	out 5 "открыть ЗДЭ02.13" <= #1228.outputOpen
	out 6 "закрыть ЗДЭ02.13" <= #1228.outputClose
	out 7 "авария открытия ЗДЭ02.13" <= #1228.errorToOpen
	#1229 OR(panTestValvesFS020201, #1230.regenFilterOUT)
	out 8 "авария закрытия ЗДЭ02.13" <= #1228.errorToClose
	#1230 FS020201manager:FilterQueueManager(input: pin 1, filterAlarm: #1231, regenFilterStatus: pin 3, alarmReset: pin 4, startNextLoop: pin 5)
	#1231 OR(alarmZD021319, pin 2, pin 11, pin 12)
	#1232 OR(#1228.errorToOpen, #1228.errorToClose, #1234.errorToOpen, #1234.errorToClose)
	#1233 alarmZD021319 <= #1232
	out 3 "ФС02.02.01 промыт" <= #1230.regenerated
	out 4 "не удалось промыть" <= #1230.failToRegen
	#1234 ZD0219:SimpleValve(inputOpen: #1229, inputClose: NOT #1229, statusOpen: pin 8, statusClose: pin 9, reset: pin 4, timeToOpenClose: pin 10)
	out 9 "открыть ЗДЭ02.19" <= #1234.outputOpen
	out 10 "закрыть ЗДЭ02.19" <= #1234.outputClose
	out 11 "авария открытия ЗДЭ02.19" <= #1234.errorToOpen
	out 12 "авария закрытия ЗДЭ02.19" <= #1234.errorToClose
END_MACRO
#1235 DD2_DO.10 <= #1227.out 2
#1236 regeneratedFS020201 <= #1227.out 3
#1237 filterFailToRegen020201 <= #1227.out 4
#1238 DD3_DO.8 <= #1227.out 5
#1239 DD3_DO.9 <= #1227.out 6
#1240 errorToOpenZD0213 <= #1227.out 7
#1241 errorToCloseZD0213 <= #1227.out 8
#1242 DD3_DO.20 <= #1227.out 9
#1243 DD3_DO.21 <= #1227.out 10
#1244 errorToOpenZD0219 <= #1227.out 11
#1245 errorToCloseZD0219 <= #1227.out 12
#1246 MACRO управление промывкой фильтра ФС02.02.02(pin 1 "сигнал на промывку": #1227.out 1, pin 2 "авария фильтра": DD7_DI.3, pin 3 "подтверждение промывки": DD7_DI.2, pin 4 "сброс аварий": alarmReset, pin 5 "начать очередь снова": filterStartNewQueue, pin 6 "ЗДЭ02.14 открыта": DD8_DI.10, pin 7 "ЗДЭ02.14 закрыта": DD8_DI.11, pin 8 "ЗДЭ02.20 открыта": DD8_DI.22, pin 9 "ЗДЭ02.20 закрыта": DD8_DI.23, pin 10 "время движения ЗДЭ": timeToOpenCloseValve, pin 11 "авария питания ЗДЭ02.14": DD9_DI.17, pin 12 "авария питания ЗДЭ02.20": DD9_DI.23)
	(* <- выход использовать в / последнем фильтре для / начала очереди заново *)
	(* если открыт = промывка *)
	(* если открыт = фильтрация *)
	out 1 "следующий в очереди" <= #1249.output
	out 2 "промыть ФС02.02.02" <= #1248
	#1247 ZD0214:SimpleValve(inputOpen: NOT #1248, inputClose: #1248, statusOpen: pin 6, statusClose: pin 7, reset: pin 4, timeToOpenClose: pin 10)
	out 5 "открыть ЗДЭ02.14" <= #1247.outputOpen
	out 6 "закрыть ЗДЭ02.14" <= #1247.outputClose
	out 7 "авария открытия ЗДЭ02.14" <= #1247.errorToOpen
	#1248 OR(panTestValvesFS020202, #1249.regenFilterOUT)
	out 8 "авария закрытия ЗДЭ02.14" <= #1247.errorToClose
	#1249 FS020202manager:FilterQueueManager(input: pin 1, filterAlarm: #1250, regenFilterStatus: pin 3, alarmReset: pin 4, startNextLoop: pin 5)
	#1250 OR(alarmZD021420, pin 2, pin 11, pin 12)
	#1251 OR(#1247.errorToOpen, #1247.errorToClose, #1253.errorToOpen, #1253.errorToClose)
	#1252 alarmZD021420 <= #1251
	out 3 "ФС02.02.02 промыт" <= #1249.regenerated
	out 4 "не удалось промыть" <= #1249.failToRegen
	#1253 ZD0220:SimpleValve(inputOpen: #1248, inputClose: NOT #1248, statusOpen: pin 8, statusClose: pin 9, reset: pin 4, timeToOpenClose: pin 10)
	out 9 "открыть ЗДЭ02.20" <= #1253.outputOpen
	out 10 "закрыть ЗДЭ02.20" <= #1253.outputClose
	out 11 "авария открытия ЗДЭ02.20" <= #1253.errorToOpen
	out 12 "авария закрытия ЗДЭ02.20" <= #1253.errorToClose
END_MACRO
#1254 DD2_DO.11 <= #1246.out 2
#1255 regeneratedFS020202 <= #1246.out 3
#1256 filterFailToRegen020202 <= #1246.out 4
#1257 DD3_DO.10 <= #1246.out 5
#1258 DD3_DO.11 <= #1246.out 6
#1259 errorToOpenZD0214 <= #1246.out 7
#1260 errorToCloseZD0214 <= #1246.out 8
#1261 DD3_DO.22 <= #1246.out 9
#1262 DD3_DO.23 <= #1246.out 10
#1263 errorToOpenZD0220 <= #1246.out 11
#1264 errorToCloseZD0220 <= #1246.out 12
#1265 MACRO управление промывкой фильтра ФС02.02.03(pin 1 "сигнал на промывку": #1246.out 1, pin 2 "авария фильтра": DD7_DI.5, pin 3 "подтверждение промывки": DD7_DI.4, pin 4 "сброс аварий": alarmReset, pin 5 "начать очередь снова": filterStartNewQueue, pin 6 "ЗДЭ02.15 открыта": DD8_DI.12, pin 7 "ЗДЭ02.15 закрыта": DD8_DI.13, pin 8 "ЗДЭ02.21 открыта": DD8_DI.24, pin 9 "ЗДЭ02.21 закрыта": DD8_DI.25, pin 10 "время движения ЗДЭ": timeToOpenCloseValve, pin 11 "авария питания ЗДЭ02.15": DD9_DI.18, pin 12 "ааврия питания ЗДЭ02.21": DD9_DI.24)
	(* <- выход использовать в / последнем фильтре для / начала очереди заново *)
	(* если открыт = промывка *)
	(* если открыт = фильтрация *)
	out 1 "следующий в очереди" <= #1268.output
	out 2 "промыть ФС02.02.03" <= #1267
	#1266 ZD0215:SimpleValve(inputOpen: NOT #1267, inputClose: #1267, statusOpen: pin 6, statusClose: pin 7, reset: pin 4, timeToOpenClose: pin 10)
	out 5 "открыть ЗДЭ02.15" <= #1266.outputOpen
	out 6 "закрыть ЗДЭ02.15" <= #1266.outputClose
	out 7 "авария открытия ЗДЭ02.15" <= #1266.errorToOpen
	#1267 OR(panTestValvesFS020203, #1268.regenFilterOUT)
	out 8 "авария закрытия ЗДЭ02.15" <= #1266.errorToClose
	#1268 FS020203manager:FilterQueueManager(input: pin 1, filterAlarm: #1269, regenFilterStatus: pin 3, alarmReset: pin 4, startNextLoop: pin 5)
	#1269 OR(alarmZD021521, pin 2, pin 11, pin 12)
	#1270 OR(#1266.errorToOpen, #1266.errorToClose, #1272.errorToOpen, #1272.errorToClose)
	#1271 alarmZD021521 <= #1270
	out 3 "ФС02.02.03 промыт" <= #1268.regenerated
	out 4 "не удалось промыть" <= #1268.failToRegen
	#1272 ZD0221:SimpleValve(inputOpen: #1267, inputClose: NOT #1267, statusOpen: pin 8, statusClose: pin 9, reset: pin 4, timeToOpenClose: pin 10)
	out 9 "открыть ЗДЭ02.21" <= #1272.outputOpen
	out 10 "закрыть ЗДЭ02.21" <= #1272.outputClose
	out 11 "авария открытия ЗДЭ02.21" <= #1272.errorToOpen
	out 12 "авария закрытия ЗДЭ02.21" <= #1272.errorToClose
END_MACRO
#1273 DD2_DO.12 <= #1265.out 2
#1274 regeneratedFS020203 <= #1265.out 3
#1275 filterFailToRegen020203 <= #1265.out 4
#1276 DD3_DO.12 <= #1265.out 5
#1277 DD3_DO.13 <= #1265.out 6
#1278 errorToOpenZD0215 <= #1265.out 7
#1279 errorToCloseZD0215 <= #1265.out 8
#1280 DD3_DO.24 <= #1265.out 9
#1281 DD3_DO.25 <= #1265.out 10
#1282 errorToOpenZD0221 <= #1265.out 11
#1283 errorToCloseZD0221 <= #1265.out 12
#1284 MACRO управление промывкой фильтра ФС02.02.04(pin 1 "сигнал на промывку": #1265.out 1, pin 2 "авария фильтра": DD7_DI.7, pin 3 "подтверждение промывки": DD7_DI.6, pin 4 "сброс аварий": alarmReset, pin 5 "начать очередь снова": filterStartNewQueue, pin 6 "ЗДЭ02.16 открыта": DD8_DI.14, pin 7 "ЗДЭ02.16 закрыта": DD8_DI.15, pin 8 "ЗДЭ02.22 открыта": DD8_DI.26, pin 9 "ЗДЭ02.22 закрыта": DD8_DI.27, pin 10 "время движения ЗДЭ": timeToOpenCloseValve, pin 11 "авария питания ЗДЭ02.16": DD9_DI.19, pin 12 "авария питания ЗДЭ02.22": DD9_DI.25)
	(* <- выход использовать в / последнем фильтре для / начала очереди заново *)
	(* если открыт = промывка *)
	(* если открыт = фильтрация *)
	out 1 "следующий в очереди" <= #1287.output
	out 2 "промыть ФС02.02.04" <= #1286
	#1285 ZD0216:SimpleValve(inputOpen: NOT #1286, inputClose: #1286, statusOpen: pin 6, statusClose: pin 7, reset: pin 4, timeToOpenClose: pin 10)
	out 5 "открыть ЗДЭ02.16" <= #1285.outputOpen
	out 6 "закрыть ЗДЭ02.16" <= #1285.outputClose
	out 7 "авария открытия ЗДЭ02.16" <= #1285.errorToOpen
	#1286 OR(panTestValvesFS020204, #1287.regenFilterOUT)
	out 8 "авария закрытия ЗДЭ02.16" <= #1285.errorToClose
	#1287 FS020204manager:FilterQueueManager(input: pin 1, filterAlarm: #1288, regenFilterStatus: pin 3, alarmReset: pin 4, startNextLoop: pin 5)
	#1288 OR(alarmZD021622, pin 2, pin 11, pin 12)
	#1289 OR(#1285.errorToOpen, #1285.errorToClose, #1291.errorToOpen, #1291.errorToClose)
	#1290 alarmZD021622 <= #1289
	out 3 "ФС02.02.04 промыт" <= #1287.regenerated
	out 4 "не удалось промыть" <= #1287.failToRegen
	#1291 ZD0222:SimpleValve(inputOpen: #1286, inputClose: NOT #1286, statusOpen: pin 8, statusClose: pin 9, reset: pin 4, timeToOpenClose: pin 10)
	out 9 "открыть ЗДЭ02.22" <= #1291.outputOpen
	out 10 "закрыть ЗДЭ02.22" <= #1291.outputClose
	out 11 "авария открытия ЗДЭ02.22" <= #1291.errorToOpen
	out 12 "авария закрытия ЗДЭ02.22" <= #1291.errorToClose
END_MACRO
#1292 DD2_DO.13 <= #1284.out 2
#1293 regeneratedFS020204 <= #1284.out 3
#1294 filterFailToRegen020204 <= #1284.out 4
#1295 DD3_DO.14 <= #1284.out 5
#1296 DD3_DO.15 <= #1284.out 6
#1297 errorToOpenZD0216 <= #1284.out 7
#1298 errorToCloseZD0216 <= #1284.out 8
#1299 DD3_DO.26 <= #1284.out 9
#1300 DD3_DO.27 <= #1284.out 10
#1301 errorToOpenZD0222 <= #1284.out 11
#1302 errorToCloseZD0222 <= #1284.out 12
#1303 MACRO управление промывкой фильтра ФС02.02.05(pin 1 "сигнал на промывку": #1284.out 1, pin 2 "авария фильтра": DD7_DI.9, pin 3 "подтверждение промывки": DD7_DI.8, pin 4 "сброс аварий": alarmReset, pin 5 "начать очередь снова": filterStartNewQueue, pin 6 "ЗДЭ02.17 открыта": DD8_DI.16, pin 7 "ЗДЭ02.17 закрыта": DD8_DI.17, pin 8 "ЗДЭ02.23 открыта": DD8_DI.28, pin 9 "ЗДЭ02.23 закрыта": DD8_DI.29, pin 10 "время движения ЗДЭ": timeToOpenCloseValve, pin 11 "авария питания ЗДЭ02.17": DD9_DI.20, pin 12 "авария питания ЗДЭ02.23": DD9_DI.26)
	(* <- выход использовать в / последнем фильтре для / начала очереди заново *)
	(* если открыт = промывка *)
	(* если открыт = фильтрация *)
	out 1 "следующий в очереди" <= #1306.output
	out 2 "промыть ФС02.02.05" <= #1305
	#1304 ZD0217:SimpleValve(inputOpen: NOT #1305, inputClose: #1305, statusOpen: pin 6, statusClose: pin 7, reset: pin 4, timeToOpenClose: pin 10)
	out 5 "открыть ЗДЭ02.17" <= #1304.outputOpen
	out 6 "закрыть ЗДЭ02.17" <= #1304.outputClose
	out 7 "авария открытия ЗДЭ02.17" <= #1304.errorToOpen
	#1305 OR(panTestValvesFS020205, #1306.regenFilterOUT)
	out 8 "авария закрытия ЗДЭ02.17" <= #1304.errorToClose
	#1306 FS020205manager:FilterQueueManager(input: pin 1, filterAlarm: #1307, regenFilterStatus: pin 3, alarmReset: pin 4, startNextLoop: pin 5)
	#1307 OR(alarmZD021723, pin 2, pin 11, pin 12)
	#1308 OR(#1304.errorToOpen, #1304.errorToClose, #1310.errorToOpen, #1310.errorToClose)
	#1309 alarmZD021723 <= #1308
	out 3 "ФС02.02.05 промыт" <= #1306.regenerated
	out 4 "не удалось промыть" <= #1306.failToRegen
	#1310 ZD0223:SimpleValve(inputOpen: #1305, inputClose: NOT #1305, statusOpen: pin 8, statusClose: pin 9, reset: pin 4, timeToOpenClose: pin 10)
	out 9 "открыть ЗДЭ02.23" <= #1310.outputOpen
	out 10 "закрыть ЗДЭ02.23" <= #1310.outputClose
	out 11 "авария открытия ЗДЭ02.23" <= #1310.errorToOpen
	out 12 "авария закрытия ЗДЭ02.23" <= #1310.errorToClose
END_MACRO
#1311 DD2_DO.14 <= #1303.out 2
#1312 regeneratedFS020205 <= #1303.out 3
#1313 filterFailToRegen020205 <= #1303.out 4
#1314 DD3_DO.16 <= #1303.out 5
#1315 DD3_DO.17 <= #1303.out 6
#1316 errorToOpenZD0217 <= #1303.out 7
#1317 errorToCloseZD0217 <= #1303.out 8
#1318 DD3_DO.28 <= #1303.out 9
#1319 DD3_DO.29 <= #1303.out 10
#1320 errorToOpenZD0223 <= #1303.out 11
#1321 errorToCloseZD0223 <= #1303.out 12
#1322 MACRO управление промывкой фильтра ФС02.02.06(pin 1 "сигнал на промывку": #1303.out 1, pin 2 "авария фильтра": DD7_DI.11, pin 3 "подтверждение промывки": DD7_DI.10, pin 4 "сброс аварий": alarmReset, pin 5 "начать очередь снова": filterStartNewQueue, pin 6 "ЗДЭ02.18 открыта": DD8_DI.18, pin 7 "ЗДЭ02.18 закрыта": DD8_DI.19, pin 8 "ЗДЭ02.24 открыта": DD8_DI.30, pin 9 "ЗДЭ02.24 закрыта": DD8_DI.31, pin 10 "время движения ЗДЭ": timeToOpenCloseValve, pin 11 "авария питания ЗДЭ02.18": DD9_DI.21, pin 12 "авария питания ЗДЭ02.24": DD9_DI.27)
	(* если открыт = промывка *)
	(* если открыт = фильтрация *)
	out 1 "промыть ФС02.02.06" <= #1324
	#1323 ZD0218:SimpleValve(inputOpen: NOT #1324, inputClose: #1324, statusOpen: pin 6, statusClose: pin 7, reset: pin 4, timeToOpenClose: pin 10)
	out 4 "открыть ЗДЭ02.18" <= #1323.outputOpen
	out 5 "закрыть ЗДЭ02.18" <= #1323.outputClose
	out 6 "авария открытия ЗДЭ02.18" <= #1323.errorToOpen
	#1324 OR(panTestValvesFS020206, #1325.regenFilterOUT)
	out 7 "авария закрытия ЗДЭ02.18" <= #1323.errorToClose
	#1325 FS020206manager:FilterQueueManager(input: pin 1, filterAlarm: #1326, regenFilterStatus: pin 3, alarmReset: pin 4, startNextLoop: pin 5)
	#1326 OR(alarmZD021824, pin 2, pin 11, pin 12)
	#1327 OR(#1323.errorToOpen, #1323.errorToClose, #1329.errorToOpen, #1329.errorToClose)
	#1328 alarmZD021824 <= #1327
	out 2 "ФС02.02.06 промыт" <= #1325.regenerated
	out 3 "не удалось промыть" <= #1325.failToRegen
	out 12 "начать очередь снова" <= #1325.regenFinished
	#1329 ZD0224:SimpleValve(inputOpen: #1324, inputClose: NOT #1324, statusOpen: pin 8, statusClose: pin 9, reset: pin 4, timeToOpenClose: pin 10)
	out 8 "открыть ЗДЭ02.24" <= #1329.outputOpen
	out 9 "закрыть ЗДЭ02.24" <= #1329.outputClose
	out 10 "авария открытия ЗДЭ02.24" <= #1329.errorToOpen
	out 11 "авария закрытия ЗДЭ02.24" <= #1329.errorToClose
END_MACRO
#1330 DD2_DO.15 <= #1322.out 1
#1331 regeneratedFS020206 <= #1322.out 2
#1332 filterFailToRegen020206 <= #1322.out 3
#1333 DD3_DO.18 <= #1322.out 4
#1334 DD3_DO.19 <= #1322.out 5
#1335 errorToOpenZD0218 <= #1322.out 6
#1336 errorToCloseZD0218 <= #1322.out 7
#1337 DD3_DO.30 <= #1322.out 8
#1338 DD3_DO.31 <= #1322.out 9
#1339 errorToOpenZD0224 <= #1322.out 10
#1340 errorToCloseZD0224 <= #1322.out 11
#1341 filterStartNewQueue <= #1322.out 12
_END_CFC_
END_PROGRAM

(* POU DosingPumpProportional, CFC *)
FUNCTION_BLOCK DosingPumpProportional
VAR_INPUT
	flowValue: REAL;		(*текущее значение мгновенного расхода, кубометров в час.*)
	setMinPumpDosingValue: REAL := 0;		(*задание минимальной производительности доз.насоса.
По умолчанию, если ничего не подключено ко входу, равно нулю.*)
	setMaxPumpDosingValue: REAL;		(*задание максимальной производительности доз.насоса, в мл/мин*)
	minOutputValue: REAL := 4;		(*минимальное значение выходного сигнала.
По умолчанию, если ничего не подключено ко входу, равно 4.*)
	maxOutputValue: REAL := 20;		(*Максимально значение выходного сигнала.
			По умолчанию, если ничего не подключено ко входу, равно 20.*)
	setKoeffProportionality: REAL;		(*Задание мл на кубометр (коэф.пропорциональности между расходом и дозированием)*)
	minFlowToStart: REAL := 10;		(*Минимальное значение расхода для подачи сигнала на начало дозирования.
			По умолчанию, если ничего не подключено ко входу, равно 10 кубометров в час.*)
END_VAR
VAR_OUTPUT
	outputValue: REAL;		(*Выходной сигнал на дозирующий насос.*)
	dosingError: BOOL;		(*Ошибка производительности дозирования (неверно заданы значения производительности насоса, производительность доз.насоса не соответствует расходу.*)
	startDosingPump: BOOL;		(*Сигнал на запуск дозирующего насоса.*)
END_VAR
VAR
	linearTransformator: LIN_TRAFO;		(*получает на вход значение из указанного диапазона, ставит на выходе пропорциональное значение из другого диапазона.*)
END_VAR
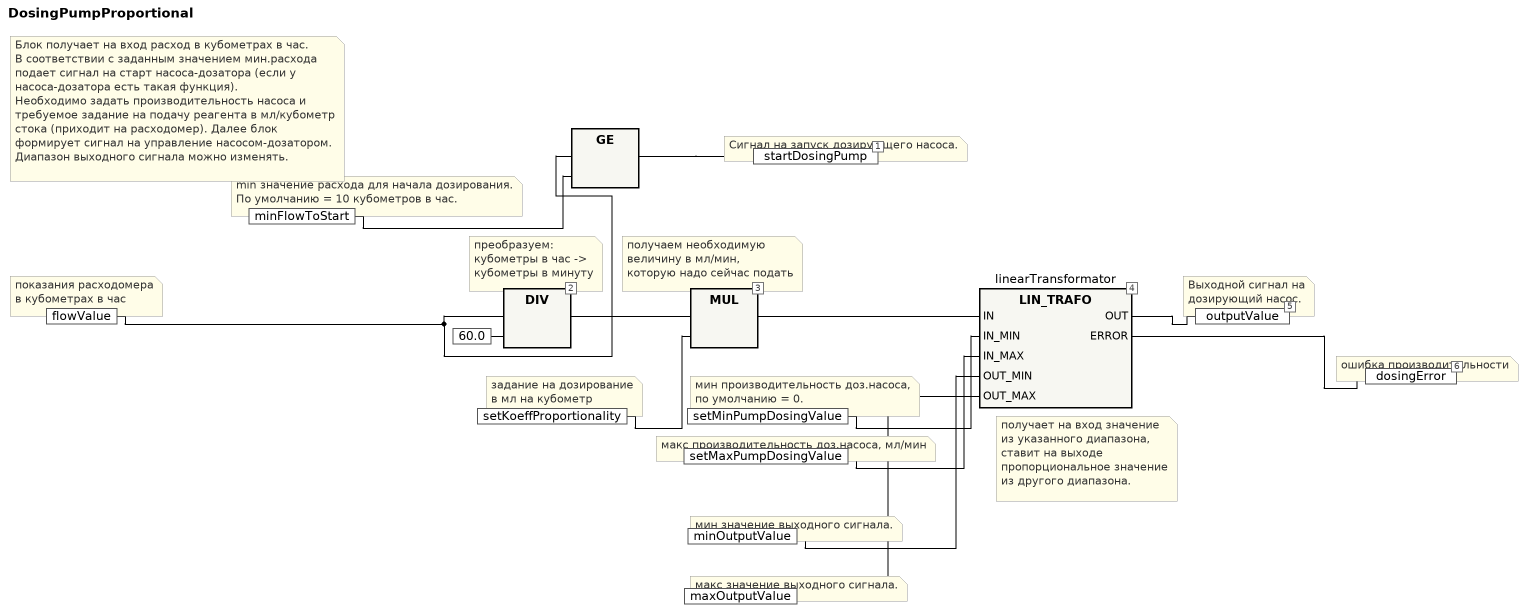
_CFC_ (* Continuous Function Chart, elements in execution order *)
(* Сигнал на запуск дозирующего насоса. *)
(* min значение расхода для начала дозирования. / По умолчанию = 10 кубометров в час. *)
(* макс производительность доз.насоса, мл/мин *)
(* мин производительность доз.насоса, / по умолчанию = 0. *)
(* получаем необходимую / величину в мл/мин, / которую надо сейчас подать *)
(* задание на дозирование / в мл на кубометр *)
(* показания расходомера / в кубометрах в час *)
(* преобразуем: / кубометры в час -> / кубометры в минуту *)
(* мин значение выходного сигнала. *)
(* макс значение выходного сигнала. *)
(* Выходной сигнал на / дозирующий насос. *)
(* ошибка производительности *)
(* получает на вход значение / из указанного диапазона, / ставит на выходе / пропорциональное значение / из другого диапазона. *)
(* Блок получает на вход расход в кубометрах в час. / В соответствии с заданным значением мин.расхода подает сигнал на старт насоса-дозатора (если у насоса-дозатора есть такая функция). / Необходимо задать производительность насоса и требуемое задание на подачу реагента в мл/кубометр стока (приходит на расходомер). Далее блок формирует сигнал на управление насосом-дозатором. / Диапазон выходного сигнала можно изменять. *)
#0 GE(flowValue, minFlowToStart)
#1 startDosingPump <= #0
#2 DIV(flowValue, 60.0)
#3 MUL(#2, setKoeffProportionality)
#4 linearTransformator:LIN_TRAFO(IN: #3, IN_MIN: setMinPumpDosingValue, IN_MAX: setMaxPumpDosingValue, OUT_MIN: minOutputValue, OUT_MAX: maxOutputValue)
#5 outputValue <= #4.OUT
#6 dosingError <= #4.ERROR
_END_CFC_
(* the same logic as Structured Text *)
(* Сигнал на запуск дозирующего насоса. *)
(* min значение расхода для начала дозирования. / По умолчанию = 10 кубометров в час. *)
(* макс производительность доз.насоса, мл/мин *)
(* мин производительность доз.насоса, / по умолчанию = 0. *)
(* получаем необходимую / величину в мл/мин, / которую надо сейчас подать *)
(* задание на дозирование / в мл на кубометр *)
(* показания расходомера / в кубометрах в час *)
(* преобразуем: / кубометры в час -> / кубометры в минуту *)
(* мин значение выходного сигнала. *)
(* макс значение выходного сигнала. *)
(* Выходной сигнал на / дозирующий насос. *)
(* ошибка производительности *)
(* получает на вход значение / из указанного диапазона, / ставит на выходе / пропорциональное значение / из другого диапазона. *)
(* Блок получает на вход расход в кубометрах в час. / В соответствии с заданным значением мин.расхода подает сигнал на старт насоса-дозатора (если у насоса-дозатора есть такая функция). / Необходимо задать производительность насоса и требуемое задание на подачу реагента в мл/кубометр стока (приходит на расходомер). Далее блок формирует сигнал на управление насосом-дозатором. / Диапазон выходного сигнала можно изменять. *)
startDosingPump := flowValue >= minFlowToStart;
linearTransformator(IN := (flowValue / 60.0) * setKoeffProportionality, IN_MIN := setMinPumpDosingValue, IN_MAX := setMaxPumpDosingValue, OUT_MIN := minOutputValue, OUT_MAX := maxOutputValue);
outputValue := linearTransformator.OUT;
dosingError := linearTransformator.ERROR;
END_FUNCTION_BLOCK

(* POU choosePumpRegime, CFC *)
FUNCTION_BLOCK choosePumpRegime
VAR
	pump1RStrig: RS;		(*Триггер-защелка выбора режима с главным первым насосом.*)
	pump2RStrig: RS;		(*Триггер-защелка выбора режима с главным вторым насосом.*)
	byCounterRStrig: RS;		(*Триггер-защелка выбора режима с запуском по количеству включений.*)
	byWorkTimeRStrig: RS;		(*Триггер-защелка выбора режима с запуском по наработке.*)
	Pump1MainDetector: R_TRIG;		(*Детектор переднего фронта включения режима, когда главный насос - первый.
			Для сброса остальных значений.*)
	Pump2MainDetector: R_TRIG;		(*Детектор переднего фронта включения режима, когда главный насос - второй.
			Для сброса остальных значений.*)
	ByCounterDetector: R_TRIG;		(*Детектор переднего фронта включения режима по количеству включений.
			Для сброса остальных значений.*)
	ByWorkTimeDetector: R_TRIG;		(*Детектор переднего фронта включения режима по наработке.
			Для сброса остальных значений.*)
END_VAR
VAR_INPUT
	start: BOOL;		(*Сигнал на включение насоса.
			Активируется выход согласно выбранного режима.*)
	pump1Main: BOOL;		(*Режим: первый насос главный, второй - резервный.*)
	pump2Main: BOOL;		(*Режим: второй насос главный, первый - резервный.*)
	byCounter: BOOL;		(*Режим: запуск по количеству включений.
			Включится с меньшим количеством стартов.*)
	byWorkTime: BOOL;		(*Режим: запуск по наработке.
			Включится насос с меньшей наработкой.*)
END_VAR
VAR_OUTPUT
	pump1MainActive: BOOL;		(*Активный режим: первый насос главный.*)
	pump2MainActive: BOOL;		(*Активный режим: второй насос главный.*)
	byCounterActive: BOOL;		(*Активный режим: включение по количеству запусков.*)
	byWorkTimeActive: BOOL;		(*Активный режим: по наработке.*)
	startPump1: BOOL;		(*Запуск первого насоса как главного (основного).*)
	startPump2: BOOL;		(*Запуск второго насоса как главного (основного).*)
	startByCounter: BOOL;		(*Запуск насоса по количеству стартов.
			Запустится с меньшим. Если одинаково, то - первый.*)
	startByWorkTime: BOOL;		(*Запуск по наработке.
			Включится с меньшей. Если одинаково, то - первый.*)
END_VAR
VAR (* helpers for the ST form of the networks *)
	_en62 : BOOL;
	_t62 : BOOL;
	_en72 : BOOL;
	_t72 : BOOL;
	_en78 : BOOL;
	_t78 : BOOL;
	_en84 : BOOL;
	_t84 : BOOL;
END_VAR
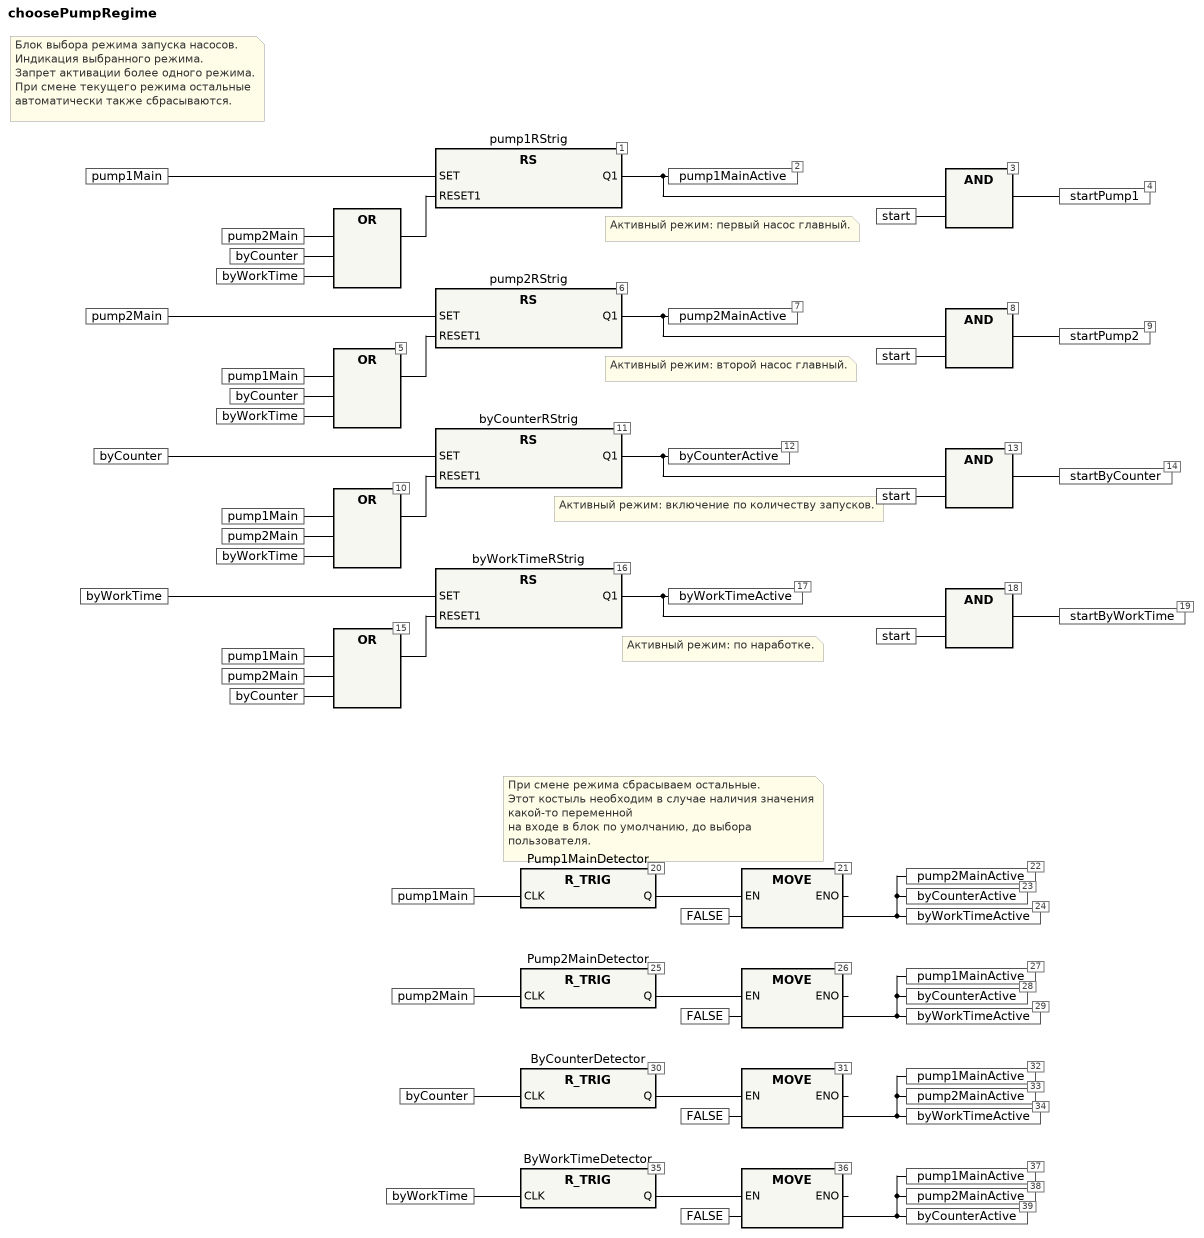
_CFC_ (* Continuous Function Chart, elements in execution order *)
(* Блок выбора режима запуска насосов. / Индикация выбранного режима. / Запрет активации более одного режима. / При смене текущего режима остальные автоматически также сбрасываются. *)
(* Активный режим: первый насос главный. *)
(* Активный режим: включение по количеству запусков. *)
(* Активный режим: по наработке. *)
(* Активный режим: второй насос главный. *)
(* При смене режима сбрасываем остальные. / Этот костыль необходим в случае наличия значения какой-то переменной / на входе в блок по умолчанию, до выбора пользователя. *)
#0 OR(pump2Main, byCounter, byWorkTime)
#1 pump1RStrig:RS(SET: pump1Main, RESET1: #0)
#2 pump1MainActive <= #1.Q1
#3 AND(#1.Q1, start)
#4 startPump1 <= #3
#5 OR(pump1Main, byCounter, byWorkTime)
#6 pump2RStrig:RS(SET: pump2Main, RESET1: #5)
#7 pump2MainActive <= #6.Q1
#8 AND(#6.Q1, start)
#9 startPump2 <= #8
#10 OR(pump1Main, pump2Main, byWorkTime)
#11 byCounterRStrig:RS(SET: byCounter, RESET1: #10)
#12 byCounterActive <= #11.Q1
#13 AND(#11.Q1, start)
#14 startByCounter <= #13
#15 OR(pump1Main, pump2Main, byCounter)
#16 byWorkTimeRStrig:RS(SET: byWorkTime, RESET1: #15)
#17 byWorkTimeActive <= #16.Q1
#18 AND(#16.Q1, start)
#19 startByWorkTime <= #18
#20 Pump1MainDetector:R_TRIG(CLK: pump1Main)
#21 MOVE(EN: #20.Q, FALSE)
#22 pump2MainActive <= #21
#23 byCounterActive <= #21
#24 byWorkTimeActive <= #21
#25 Pump2MainDetector:R_TRIG(CLK: pump2Main)
#26 MOVE(EN: #25.Q, FALSE)
#27 pump1MainActive <= #26
#28 byCounterActive <= #26
#29 byWorkTimeActive <= #26
#30 ByCounterDetector:R_TRIG(CLK: byCounter)
#31 MOVE(EN: #30.Q, FALSE)
#32 pump1MainActive <= #31
#33 pump2MainActive <= #31
#34 byWorkTimeActive <= #31
#35 ByWorkTimeDetector:R_TRIG(CLK: byWorkTime)
#36 MOVE(EN: #35.Q, FALSE)
#37 pump1MainActive <= #36
#38 pump2MainActive <= #36
#39 byCounterActive <= #36
_END_CFC_
(* the same logic as Structured Text *)
(* Блок выбора режима запуска насосов. / Индикация выбранного режима. / Запрет активации более одного режима. / При смене текущего режима остальные автоматически также сбрасываются. *)
(* Активный режим: первый насос главный. *)
(* Активный режим: включение по количеству запусков. *)
(* Активный режим: по наработке. *)
(* Активный режим: второй насос главный. *)
(* При смене режима сбрасываем остальные. / Этот костыль необходим в случае наличия значения какой-то переменной / на входе в блок по умолчанию, до выбора пользователя. *)
pump1RStrig(SET := pump1Main, RESET1 := pump2Main OR byCounter OR byWorkTime);
pump1MainActive := pump1RStrig.Q1;
startPump1 := pump1RStrig.Q1 AND start;
pump2RStrig(SET := pump2Main, RESET1 := pump1Main OR byCounter OR byWorkTime);
pump2MainActive := pump2RStrig.Q1;
startPump2 := pump2RStrig.Q1 AND start;
byCounterRStrig(SET := byCounter, RESET1 := pump1Main OR pump2Main OR byWorkTime);
byCounterActive := byCounterRStrig.Q1;
startByCounter := byCounterRStrig.Q1 AND start;
byWorkTimeRStrig(SET := byWorkTime, RESET1 := pump1Main OR pump2Main OR byCounter);
byWorkTimeActive := byWorkTimeRStrig.Q1;
startByWorkTime := byWorkTimeRStrig.Q1 AND start;
Pump1MainDetector(CLK := pump1Main);
_en62 := Pump1MainDetector.Q;
IF _en62 THEN _t62 := FALSE; END_IF;
IF _en62 THEN pump2MainActive := _t62; END_IF;
IF _en62 THEN byCounterActive := _t62; END_IF;
IF _en62 THEN byWorkTimeActive := _t62; END_IF;
Pump2MainDetector(CLK := pump2Main);
_en72 := Pump2MainDetector.Q;
IF _en72 THEN _t72 := FALSE; END_IF;
IF _en72 THEN pump1MainActive := _t72; END_IF;
IF _en72 THEN byCounterActive := _t72; END_IF;
IF _en72 THEN byWorkTimeActive := _t72; END_IF;
ByCounterDetector(CLK := byCounter);
_en78 := ByCounterDetector.Q;
IF _en78 THEN _t78 := FALSE; END_IF;
IF _en78 THEN pump1MainActive := _t78; END_IF;
IF _en78 THEN pump2MainActive := _t78; END_IF;
IF _en78 THEN byWorkTimeActive := _t78; END_IF;
ByWorkTimeDetector(CLK := byWorkTime);
_en84 := ByWorkTimeDetector.Q;
IF _en84 THEN _t84 := FALSE; END_IF;
IF _en84 THEN pump1MainActive := _t84; END_IF;
IF _en84 THEN pump2MainActive := _t84; END_IF;
IF _en84 THEN byCounterActive := _t84; END_IF;
END_FUNCTION_BLOCK

(* POU TwoPumpManager, CFC *)
FUNCTION_BLOCK TwoPumpManager
VAR_INPUT
	startStopPump1: BOOL;		(*Сигнал на пуск/стоп первого насоса.*)
	startStopPump2: BOOL;		(*Сигнал на пуск/стоп второго насоса.*)
	alarmPump1: BOOL;		(*Сигнал "авария" на первом насосе.*)
	alarmPump2: BOOL;		(*Сигнал "авария" на втором насосе.*)
	alarmReset: BOOL;		(*Сброс аварии.*)

	counterStart: BOOL;		(*Запуск насоса с меньшим количеством включений.*)
	Pump1ResetCounter: BOOL;		(*Сброс счетчика количества включений первого насоса.
Сбрасывается также автоматически при достижении счетчиком значения ValueToResetCTU.*)
	Pump2ResetCounter: BOOL;		(*Сброс счетчика количества включений второго насоса.
Сбрасывается также автоматически при достижении счетчиком значения ValueToResetCTU.*)
	ValueToResetCounter: WORD := 32767;		(*Значение счетчика, после которого он сбрасывается на ноль.
			Максимальное допустимое значение: 32767, будет установлено, если не подключать ничего на вход.*)

	workTimeStart: BOOL;		(*Запуск насоса с выбором по меньшей наработке.*)
	workTimePump1Reset: BOOL;		(*Сброс времени наработки первого насоса.*)
	workTimePump2Reset: BOOL;		(*Сброс времени наработки второго насоса.*)
END_VAR
VAR_OUTPUT
	pump1ON: BOOL;		(*Выход на включение первого насоса.*)
	pump2ON: BOOL;		(*Выход на включение второго насоса.*)

	counterPump1: WORD;		(*Количество включений первого насоса.
При достижении значения ValueToResetCTU сбрасывается в ноль.*)
	counterPump2: WORD;		(*Количество включений второго насоса.
При достижении значения ValueToResetCTU сбрасывается в ноль.*)

	currentWorkTimePump1: DWORD;		(*Текущая наработка первого насоса.*)
	currentWorkTimePump2: DWORD;		(*Текущая наработка второго насоса.*)
END_VAR
VAR
	RtrigPump1: R_TRIG;		(*Включает первый насос по фронту сигнала на ручной пуск/стоп.*)
	FtrigPump1: F_TRIG;		(*Выключает первый насос по спаду сигнала на ручной пуск/стоп.*)
	RtrigPump2: R_TRIG;		(*Включает второй насос по фронту сигнала на ручной пуск/стоп.*)
	FtrigPump2: F_TRIG;		(*Выключает второй насос по спаду сигнала на ручной пуск/стоп.*)
	RSpump1: RS;		(*RS-триггер нормального включения первого насоса*)
	RSpump2: RS;		(*RS-триггер нормального включения второго насоса*)
	pump1NormalON: BOOL;		(*Сигнал нормального (неаварийного) включения первого насоса.*)
	pump2NormalON: BOOL;		(*Сигнал нормального (неаварийного) включения второго насоса.*)
	pump2EmergencyON: BOOL;		(*Сигнал аварийного включения второго насоса (при аварии первого).*)
	pump1EmergencyON: BOOL;		(*Сигнал аварийного включения первого насоса (при аварии второго).*)
	alarmPump1RStrig: RS;		(*Триггер аварии первого насоса.*)
	alarmPump2RStrig: RS;		(*Триггер аварии второго насоса.*)
	TONtoOnPump1: TON;		(*Таймер задержки включения первого насоса, на переключение контакторов при аварийном переключении.
			Жестко задано 1 секунда.*)
	TONtoOnPump2: TON;		(*Таймер задержки включения второго насоса, на переключение контакторов при аварийном переключении.
						Жестко задано 1 секунда.*)

	CTUPump1: CTU;		(*Счетчик количества включений первого насоса.*)
	CTUPump2: CTU;		(*Счетчик количества включений второго насоса.*)
	counterRtrig: R_TRIG;		(*Детектор переднего фронта сигнала на старт насоса с меньшей наработкой, включает насос.*)
	counterFtrig: F_TRIG;		(*Детектор спада сигнала на запуск насоса с меньшей наработкой, останавливает насос.*)
	counterRStrigPump1: RS;		(*Триггер-защелка включения первого насоса при запуске по количеству включений.*)
	counterRStrigPump2: RS;		(*Триггер-защелка включения второго насоса при запуске по количеству включений.*)
	counterPump1ON: BOOL;		(*Сигнал на запуск первого насоса при запуске по количеству включений.*)
	counterPump2ON: BOOL;		(*Сигнал на запуск второго насоса при запуске по количеству включений.*)

	workTimePump1ON: BOOL;		(*Сигнал на запуск первого насоса при запуске по наработке.*)
	workTimePump2ON: BOOL;		(*Сигнал на запуск второго насоса при запуске по наработке.*)
	timeStartFtrig: F_TRIG;		(*Детектор спада сигнала на запуск по наработке.*)
	timeStartRtrig: R_TRIG;		(*Детектор переднего фронта сигнала на запуск по наработке.*)
	RStrigTimePump1: RS;		(*Триггер-защелка запуск первого насоса по наработке.*)
	RStrigTimePump2: RS;		(*Триггер-защелка запуск второго насоса по наработке.*)

	pulsarP1: PulsePerSec; (* генератор импульса в секунду для наработки 1 насоса*)
	pulsarP2: PulsePerSec; (* генератор импульса в секунду для наработки 2 насоса*)


END_VAR
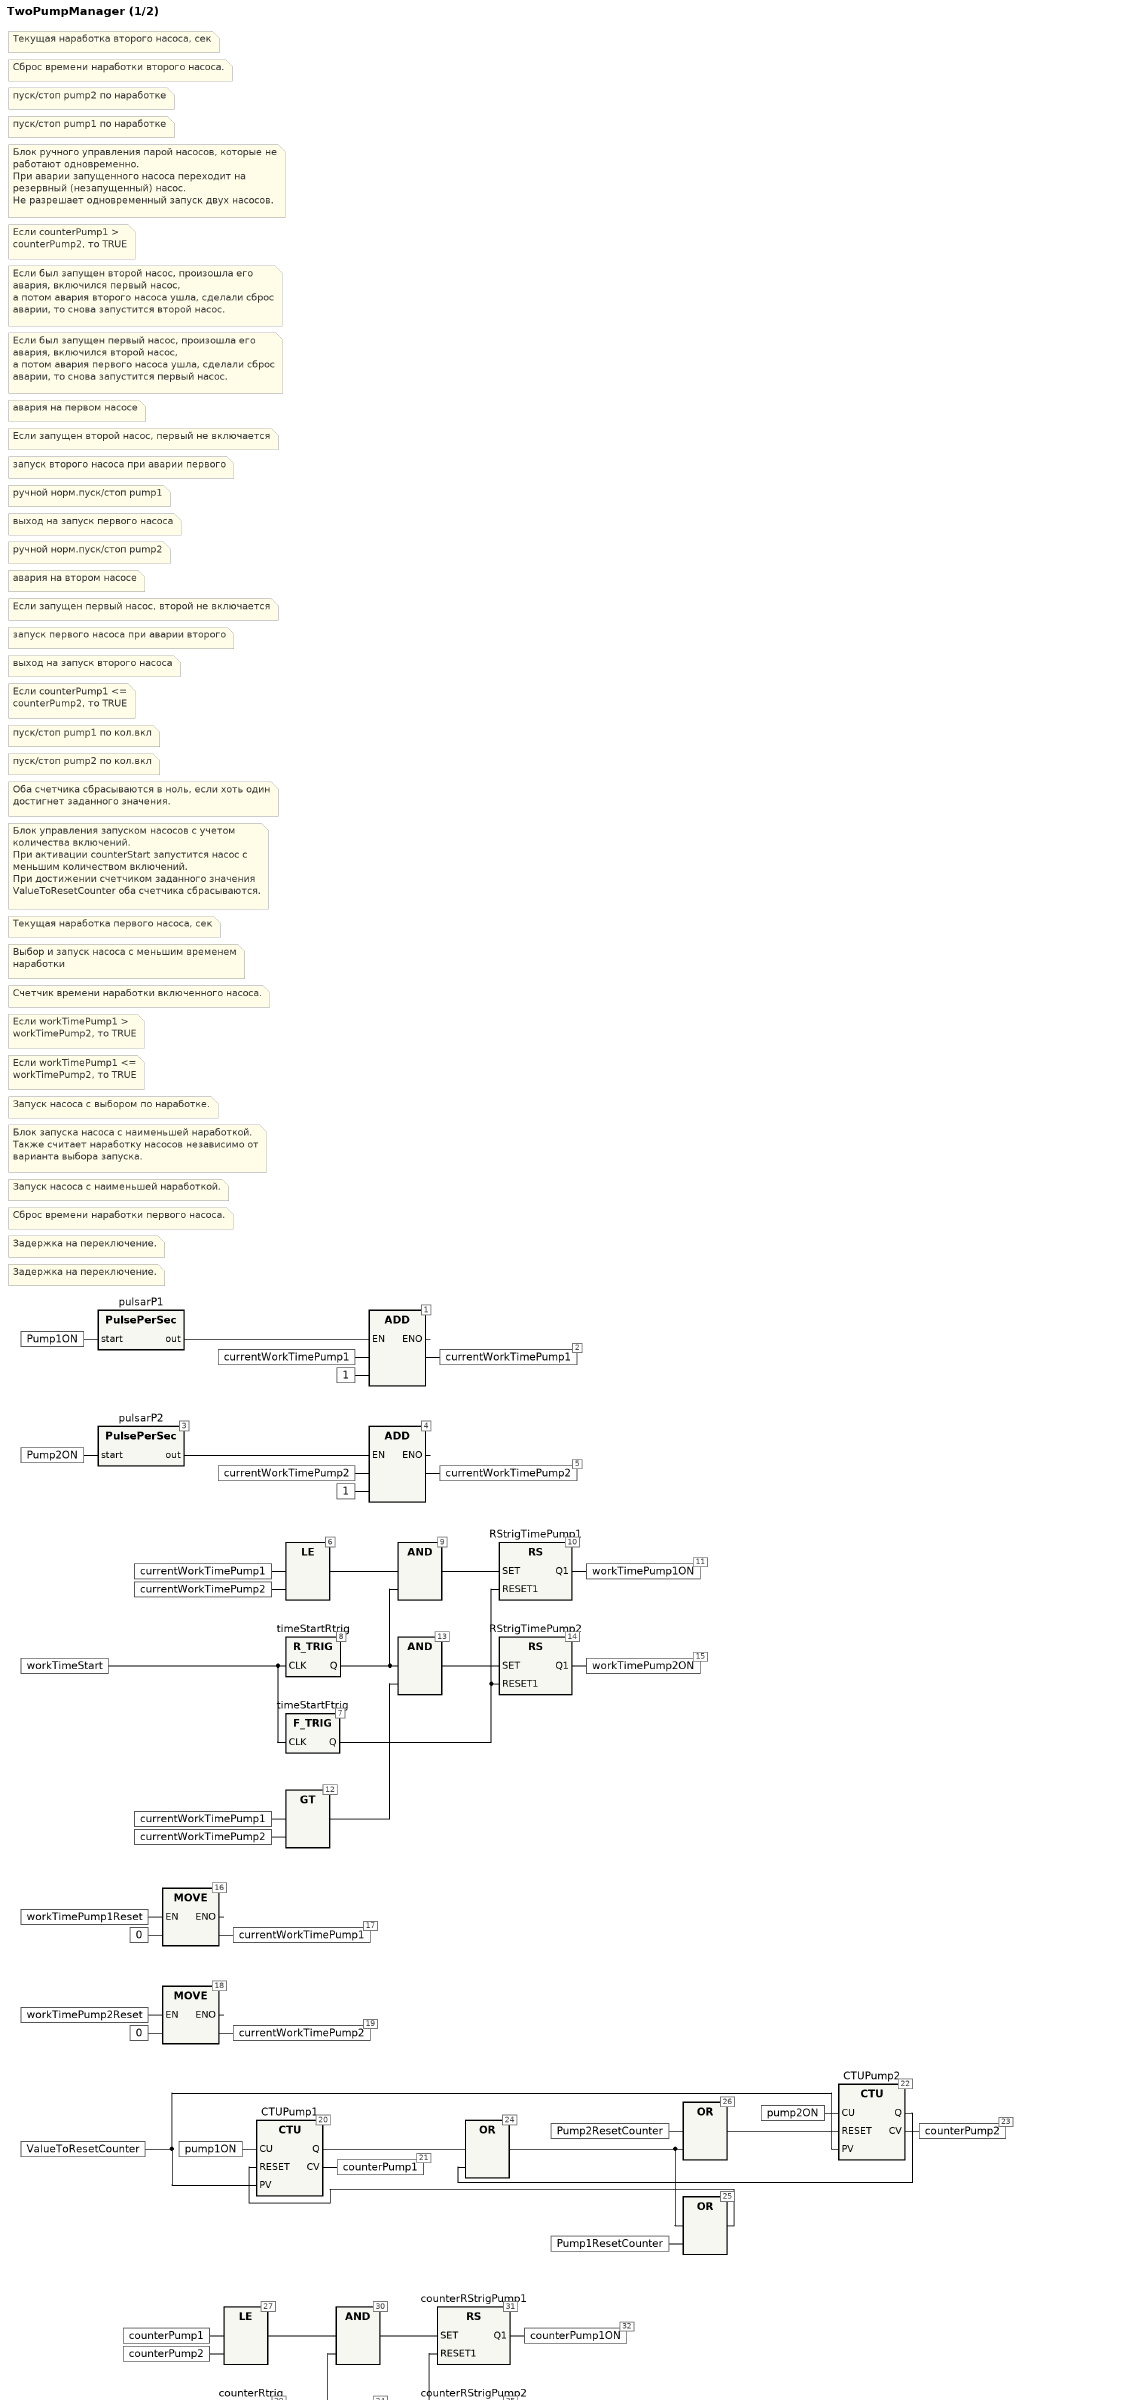
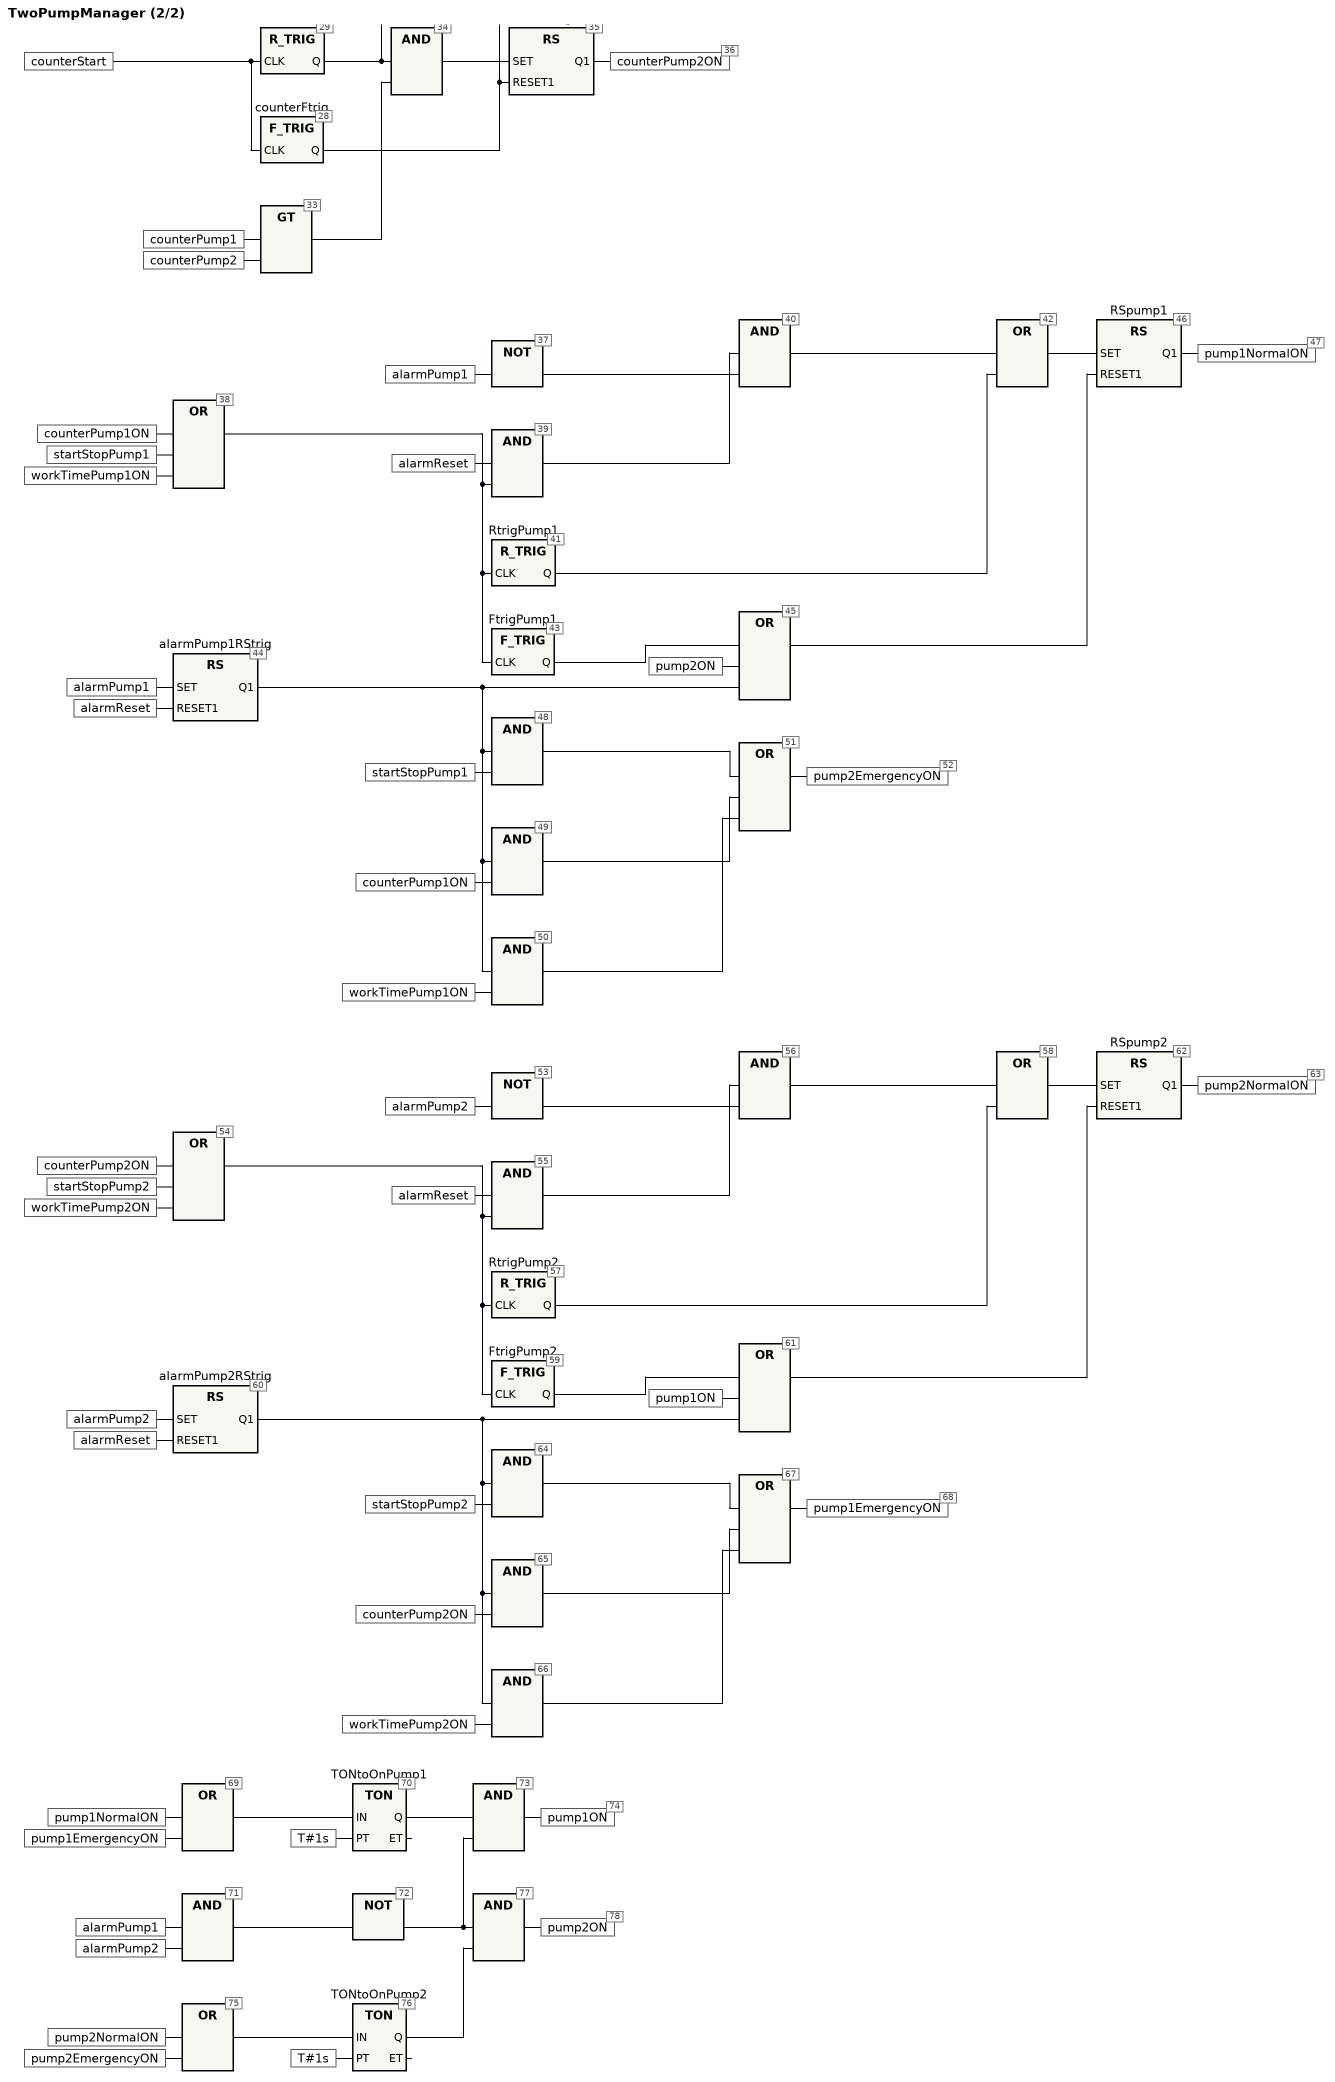
_CFC_ (* Continuous Function Chart, elements in execution order *)
(* Текущая наработка второго насоса, сек *)
(* Сброс времени наработки второго насоса. *)
(* пуск/стоп pump2 по наработке *)
(* пуск/стоп pump1 по наработке *)
(* Блок ручного управления парой насосов, которые не работают одновременно. / При аварии запущенного насоса переходит на резервный (незапущенный) насос. / Не разрешает одновременный запуск двух насосов. *)
(* Если counterPump1 > / counterPump2, то TRUE *)
(* Если был запущен второй насос, произошла его авария, включился первый насос, / а потом авария второго насоса ушла, сделали сброс аварии, то снова запустится второй насос. *)
(* Если был запущен первый насос, произошла его авария, включился второй насос, / а потом авария первого насоса ушла, сделали сброс аварии, то снова запустится первый насос. *)
(* авария на первом насосе *)
(* Если запущен второй насос, первый не включается *)
(* запуск второго насоса при аварии первого *)
(* ручной норм.пуск/стоп pump1 *)
(* выход на запуск первого насоса *)
(* ручной норм.пуск/стоп pump2 *)
(* авария на втором насосе *)
(* Если запущен первый насос, второй не включается *)
(* запуск первого насоса при аварии второго *)
(* выход на запуск второго насоса *)
(* Если counterPump1 <= / counterPump2, то TRUE *)
(* пуск/стоп pump1 по кол.вкл *)
(* пуск/стоп pump2 по кол.вкл *)
(* Оба счетчика сбрасываются в ноль, если хоть один достигнет заданного значения. *)
(* Блок управления запуском насосов с учетом количества включений. / При активации counterStart запустится насос с меньшим количеством включений. / При достижении счетчиком заданного значения ValueToResetCounter оба счетчика сбрасываются. *)
(* Текущая наработка первого насоса, сек *)
(* Выбор и запуск насоса с меньшим временем наработки *)
(* Счетчик времени наработки включенного насоса. *)
(* Если workTimePump1 > / workTimePump2, то TRUE *)
(* Если workTimePump1 <= / workTimePump2, то TRUE *)
(* Запуск насоса с выбором по наработке. *)
(* Блок запуска насоса с наименьшей наработкой. / Также считает наработку насосов независимо от варианта выбора запуска. *)
(* Запуск насоса с наименьшей наработкой. *)
(* Сброс времени наработки первого насоса. *)
(* Задержка на переключение. *)
(* Задержка на переключение. *)
#0 pulsarP1:PulsePerSec(start: Pump1ON)
#1 ADD(EN: #0.out, currentWorkTimePump1, 1)
#2 currentWorkTimePump1 <= #1
#3 pulsarP2:PulsePerSec(start: Pump2ON)
#4 ADD(EN: #3.out, currentWorkTimePump2, 1)
#5 currentWorkTimePump2 <= #4
#6 LE(currentWorkTimePump1, currentWorkTimePump2)
#7 timeStartFtrig:F_TRIG(CLK: workTimeStart)
#8 timeStartRtrig:R_TRIG(CLK: workTimeStart)
#9 AND(#6, #8.Q)
#10 RStrigTimePump1:RS(SET: #9, RESET1: #7.Q)
#11 workTimePump1ON <= #10.Q1
#12 GT(currentWorkTimePump1, currentWorkTimePump2)
#13 AND(#8.Q, #12)
#14 RStrigTimePump2:RS(SET: #13, RESET1: #7.Q)
#15 workTimePump2ON <= #14.Q1
#16 MOVE(EN: workTimePump1Reset, 0)
#17 currentWorkTimePump1 <= #16
#18 MOVE(EN: workTimePump2Reset, 0)
#19 currentWorkTimePump2 <= #18
#20 CTUPump1:CTU(CU: pump1ON, RESET: #25, PV: ValueToResetCounter)
#21 counterPump1 <= #20.CV
#22 CTUPump2:CTU(CU: pump2ON, RESET: #26, PV: ValueToResetCounter)
#23 counterPump2 <= #22.CV
#24 OR(#20.Q, #22.Q)
#25 OR(#24, Pump1ResetCounter)
#26 OR(Pump2ResetCounter, #24)
#27 LE(counterPump1, counterPump2)
#28 counterFtrig:F_TRIG(CLK: counterStart)
#29 counterRtrig:R_TRIG(CLK: counterStart)
#30 AND(#27, #29.Q)
#31 counterRStrigPump1:RS(SET: #30, RESET1: #28.Q)
#32 counterPump1ON <= #31.Q1
#33 GT(counterPump1, counterPump2)
#34 AND(#29.Q, #33)
#35 counterRStrigPump2:RS(SET: #34, RESET1: #28.Q)
#36 counterPump2ON <= #35.Q1
#37 NOT(alarmPump1)
#38 OR(counterPump1ON, startStopPump1, workTimePump1ON)
#39 AND(alarmReset, #38)
#40 AND(#39, #37)
#41 RtrigPump1:R_TRIG(CLK: #38)
#42 OR(#40, #41.Q)
#43 FtrigPump1:F_TRIG(CLK: #38)
#44 alarmPump1RStrig:RS(SET: alarmPump1, RESET1: alarmReset)
#45 OR(#43.Q, pump2ON, #44.Q1)
#46 RSpump1:RS(SET: #42, RESET1: #45)
#47 pump1NormalON <= #46.Q1
#48 AND(#44.Q1, startStopPump1)
#49 AND(#44.Q1, counterPump1ON)
#50 AND(#44.Q1, workTimePump1ON)
#51 OR(#48, #49, #50)
#52 pump2EmergencyON <= #51
#53 NOT(alarmPump2)
#54 OR(counterPump2ON, startStopPump2, workTimePump2ON)
#55 AND(alarmReset, #54)
#56 AND(#55, #53)
#57 RtrigPump2:R_TRIG(CLK: #54)
#58 OR(#56, #57.Q)
#59 FtrigPump2:F_TRIG(CLK: #54)
#60 alarmPump2RStrig:RS(SET: alarmPump2, RESET1: alarmReset)
#61 OR(#59.Q, pump1ON, #60.Q1)
#62 RSpump2:RS(SET: #58, RESET1: #61)
#63 pump2NormalON <= #62.Q1
#64 AND(#60.Q1, startStopPump2)
#65 AND(#60.Q1, counterPump2ON)
#66 AND(#60.Q1, workTimePump2ON)
#67 OR(#64, #65, #66)
#68 pump1EmergencyON <= #67
#69 OR(pump1NormalON, pump1EmergencyON)
#70 TONtoOnPump1:TON(IN: #69, PT: T#1s)
#71 AND(alarmPump1, alarmPump2)
#72 NOT(#71)
#73 AND(#70.Q, #72)
#74 pump1ON <= #73
#75 OR(pump2NormalON, pump2EmergencyON)
#76 TONtoOnPump2:TON(IN: #75, PT: T#1s)
#77 AND(#72, #76.Q)
#78 pump2ON <= #77
_END_CFC_
END_FUNCTION_BLOCK

(* POU PulsePerSec, CFC *)
FUNCTION_BLOCK PulsePerSec
VAR_INPUT
	start: BOOL;		(*Включает генератор импульсов.*)
END_VAR
VAR_OUTPUT
	out: BOOL;		(*Выход генератора импульсов. Начинает с FALSE.
			Каждую секунду выдает BOOL: TRUE.*)
END_VAR
VAR
	sessionTime: DWORD;		(*Внутренняя переменная.
			Хранит время сессии работы генератора импульсов.*)
	sessionVariable: DWORD;		(*Внутренняя переменная. Хранит значение, отличающееся от
			переменной хранения времени сессии на единицу.*)
	pulserRtrig: R_TRIG;		(*Детектор переднего фронта подачи импульсов.*)
	pulserRTC: RTC;		(*Таймер реального времени.
			*)
END_VAR
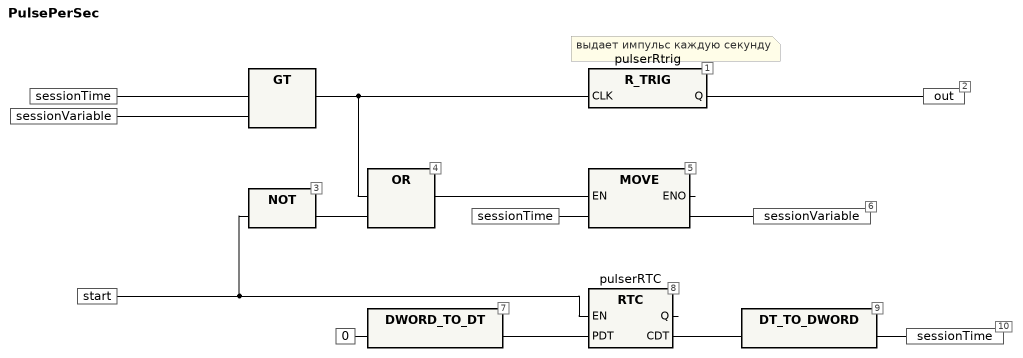
_CFC_ (* Continuous Function Chart, elements in execution order *)
(* выдает импульс каждую секунду *)
#0 GT(sessionTime, sessionVariable)
#1 pulserRtrig:R_TRIG(CLK: #0)
#2 out <= #1.Q
#3 NOT(start)
#4 OR(#0, #3)
#5 MOVE(EN: #4, sessionTime)
#6 sessionVariable <= #5
#7 DWORD_TO_DT(0)
#8 pulserRTC:RTC(EN: start, PDT: #7)
#9 DT_TO_DWORD(#8.CDT)
#10 sessionTime <= #9
_END_CFC_
END_FUNCTION_BLOCK

(* POU TwoPumpOneDriveManager, CFC *)
FUNCTION_BLOCK TwoPumpOneDriveManager
VAR_INPUT
	startStopPump1: BOOL;		(*Сигнал на пуск/стоп первого насоса.*)
	startStopPump2: BOOL;		(*Сигнал на пуск/стоп второго насоса.*)
	alarmPump1: BOOL;		(*Сигнал "авария" на первом насосе.*)
	alarmPump2: BOOL;		(*Сигнал "авария" на втором насосе.*)
	alarmReset: BOOL;		(*Сброс аварии.*)

	counterStart: BOOL;		(*Запуск насоса с меньшим количеством включений.*)
	Pump1ResetCounter: BOOL;		(*Сброс счетчика количества включений первого насоса.
Сбрасывается также автоматически при достижении счетчиком значения ValueToResetCTU.*)
	Pump2ResetCounter: BOOL;		(*Сброс счетчика количества включений второго насоса.
Сбрасывается также автоматически при достижении счетчиком значения ValueToResetCTU.*)
	ValueToResetCounter: WORD := 32767;		(*Значение счетчика, после которого он сбрасывается на ноль.
			Максимальное допустимое значение: 32767, будет установлено, если не подключать ничего на вход.*)

	workTimeStart: BOOL;		(*Запуск насоса с выбором по меньшей наработке.*)
	workTimePump1Reset: BOOL;		(*Сброс времени наработки первого насоса.*)
	workTimePump2Reset: BOOL;		(*Сброс времени наработки второго насоса.*)
	timeKM1off: TIME := T#20s;		(*Время на которое отключается питание ЧРП.
			По умолчанию = 20сек.*)
	timeKM23DelayON: TIME := T#15s;		(*Время задержки включения контактора насоса.
			По умолчанию = 15 сек.*)
	timeKM23offDelay: TIME := T#10s;		(*Время задержки выключения контактора насосов.
			По умолчанию = 10сек. (Чтобы сначала отключилось питание ЧРП).*)
	timeReadyToStartDelay: TIME := T#5s;		(*Время задержки подачи сигнала на старт ЧРП.
			По умолчанию = 5сек.*)
END_VAR
VAR_OUTPUT

	counterPump1: WORD;		(*Количество включений первого насоса.
При достижении значения ValueToResetCTU сбрасывается в ноль.*)
	counterPump2: WORD;		(*Количество включений второго насоса.
При достижении значения ValueToResetCTU сбрасывается в ноль.*)

	currentWorkTimePump1: DWORD;		(*Текущая наработка первого насоса.*)
	currentWorkTimePump2: DWORD;		(*Текущая наработка второго насоса.*)

	DriveKM: BOOL;		(*Выход на включение контактора частотного преобразователя (питание).*)
	pump1KM: BOOL;		(*Выход на включение контактора первого насоса.*)
	pump2KM: BOOL;		(*Выход на включение контактора второго насоса.*)
	driveStart: BOOL;		(*Сигнал на старт частотного преобразователя.*)
	pump1active: BOOL;		(*Идет процесс запуска насоса 1.*)
	pump2active: BOOL;		(*Идет процесс запуска насоса 2.*)
END_VAR
VAR
	RtrigPump1: R_TRIG;		(*Включает первый насос по фронту сигнала на ручной пуск/стоп.*)
	FtrigPump1: F_TRIG;		(*Выключает первый насос по спаду сигнала на ручной пуск/стоп.*)
	RtrigPump2: R_TRIG;		(*Включает второй насос по фронту сигнала на ручной пуск/стоп.*)
	FtrigPump2: F_TRIG;		(*Выключает второй насос по спаду сигнала на ручной пуск/стоп.*)
	RSpump1: RS;		(*RS-триггер нормального включения первого насоса*)
	RSpump2: RS;		(*RS-триггер нормального включения второго насоса*)
	pump1NormalON: BOOL;		(*Сигнал нормального (неаварийного) включения первого насоса.*)
	pump2NormalON: BOOL;		(*Сигнал нормального (неаварийного) включения второго насоса.*)
	pump2EmergencyON: BOOL;		(*Сигнал аварийного включения второго насоса (при аварии первого).*)
	pump1EmergencyON: BOOL;		(*Сигнал аварийного включения первого насоса (при аварии второго).*)
	alarmPump1RStrig: RS;		(*Триггер аварии первого насоса.*)
	alarmPump2RStrig: RS;		(*Триггер аварии второго насоса.*)
	TONtoOnPump1: TON;		(*Таймер задержки включения первого насоса, на переключение контакторов при аварийном переключении.
			Жестко задано 1 секунда.*)
	TONtoOnPump2: TON;		(*Таймер задержки включения второго насоса, на переключение контакторов при аварийном переключении.
						Жестко задано 1 секунда.*)

	CTUPump1: CTU;		(*Счетчик количества включений первого насоса.*)
	CTUPump2: CTU;		(*Счетчик количества включений второго насоса.*)
	counterRtrig: R_TRIG;		(*Детектор переднего фронта сигнала на старт насоса с меньшей наработкой, включает насос.*)
	counterFtrig: F_TRIG;		(*Детектор спада сигнала на запуск насоса с меньшей наработкой, останавливает насос.*)
	counterRStrigPump1: RS;		(*Триггер-защелка включения первого насоса при запуске по количеству включений.*)
	counterRStrigPump2: RS;		(*Триггер-защелка включения второго насоса при запуске по количеству включений.*)
	counterPump1ON: BOOL;		(*Сигнал на запуск первого насоса при запуске по количеству включений.*)
	counterPump2ON: BOOL;		(*Сигнал на запуск второго насоса при запуске по количеству включений.*)

	workTimePump1ON: BOOL;		(*Сигнал на запуск первого насоса при запуске по наработке.*)
	workTimePump2ON: BOOL;		(*Сигнал на запуск второго насоса при запуске по наработке.*)
	timeStartFtrig: F_TRIG;		(*Детектор спада сигнала на запуск по наработке.*)
	timeStartRtrig: R_TRIG;		(*Детектор переднего фронта сигнала на запуск по наработке.*)
	RStrigTimePump1: RS;		(*Триггер-защелка запуск первого насоса по наработке.*)
	RStrigTimePump2: RS;		(*Триггер-защелка запуск второго насоса по наработке.*)

	pulsarP1: PulsePerSec; (*Генератор импульсов каждую секунду для насоса 1*)
	pulsarP2: PulsePerSec; (*Генератор импульсов каждую секунду для насоса 2*)


	pump1ON: BOOL;		(*Выход на включение первого насоса.*)
	pump2ON: BOOL;		(*Выход на включение второго насоса.*)
	rTrigPump1ON: R_TRIG;		(*Детектор переднего фронта на запуск насоса 1.*)
	rTrigPump2ON: R_TRIG;		(*Детектор переднего фрона на запуск насоса 2.*)
	rTrigKM1off: R_TRIG;		(*Детектор переднего фронта сигнала на запуск одного из насосов,
			для выключения контактора КМ1 питающего ЧРП.*)
	rsTrigKM1: RS;		(*Триггер управления КМ1 (питание ЧРП).*)
	rsTrigKMpump1: RS;		(*Триггер контактора насоса 1.*)
	rsTrigKMpump2: RS;		(*Триггер контактора насоса 2.*)
	timerKM1off: TOF;		(*Таймер выключения контактора питания ЧРП.*)
	timerKM2DelayON: TON;		(*Таймер задержки включения контактора насоса 1.*)
	timerKM3DelayON: TON;		(*Таймер задержки включения контактора насоса 2.*)
	timerKM2DelayOFF: TOF;		(*Таймер задержки выключения контактора насоса 1.*)
	timerKM3DelayOFF: TOF;		(*Таймер задержки выключения контактора насоса 2.*)
	timerReadyToStartON: TON;		(*Таймер задержки подачи сигнала о готовности к старту (запуск ЧРП).*)
END_VAR
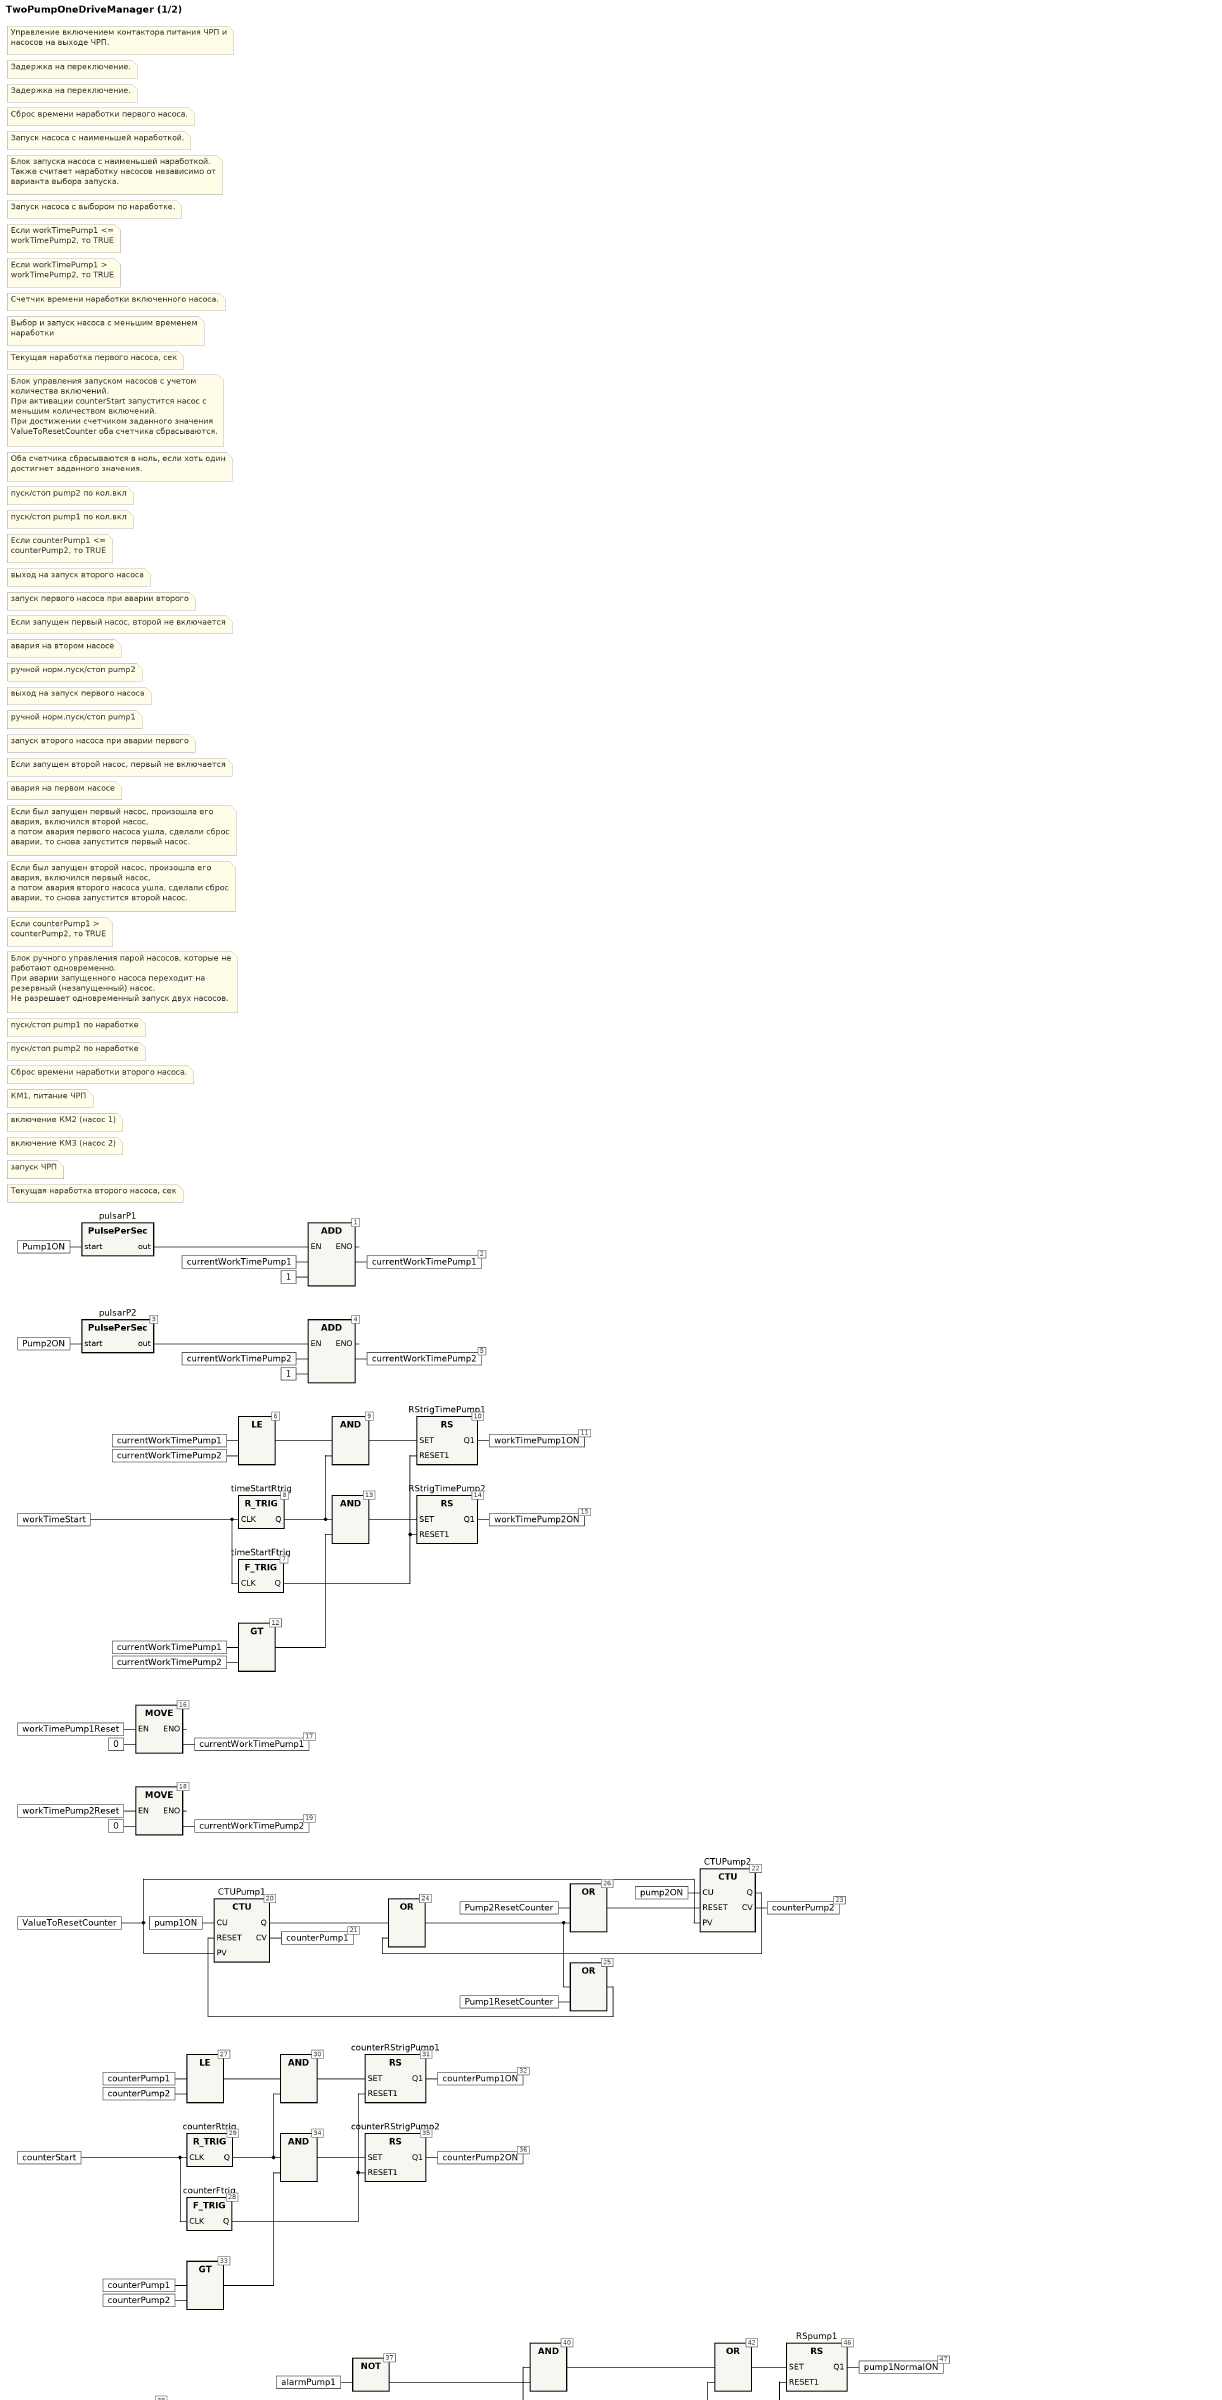
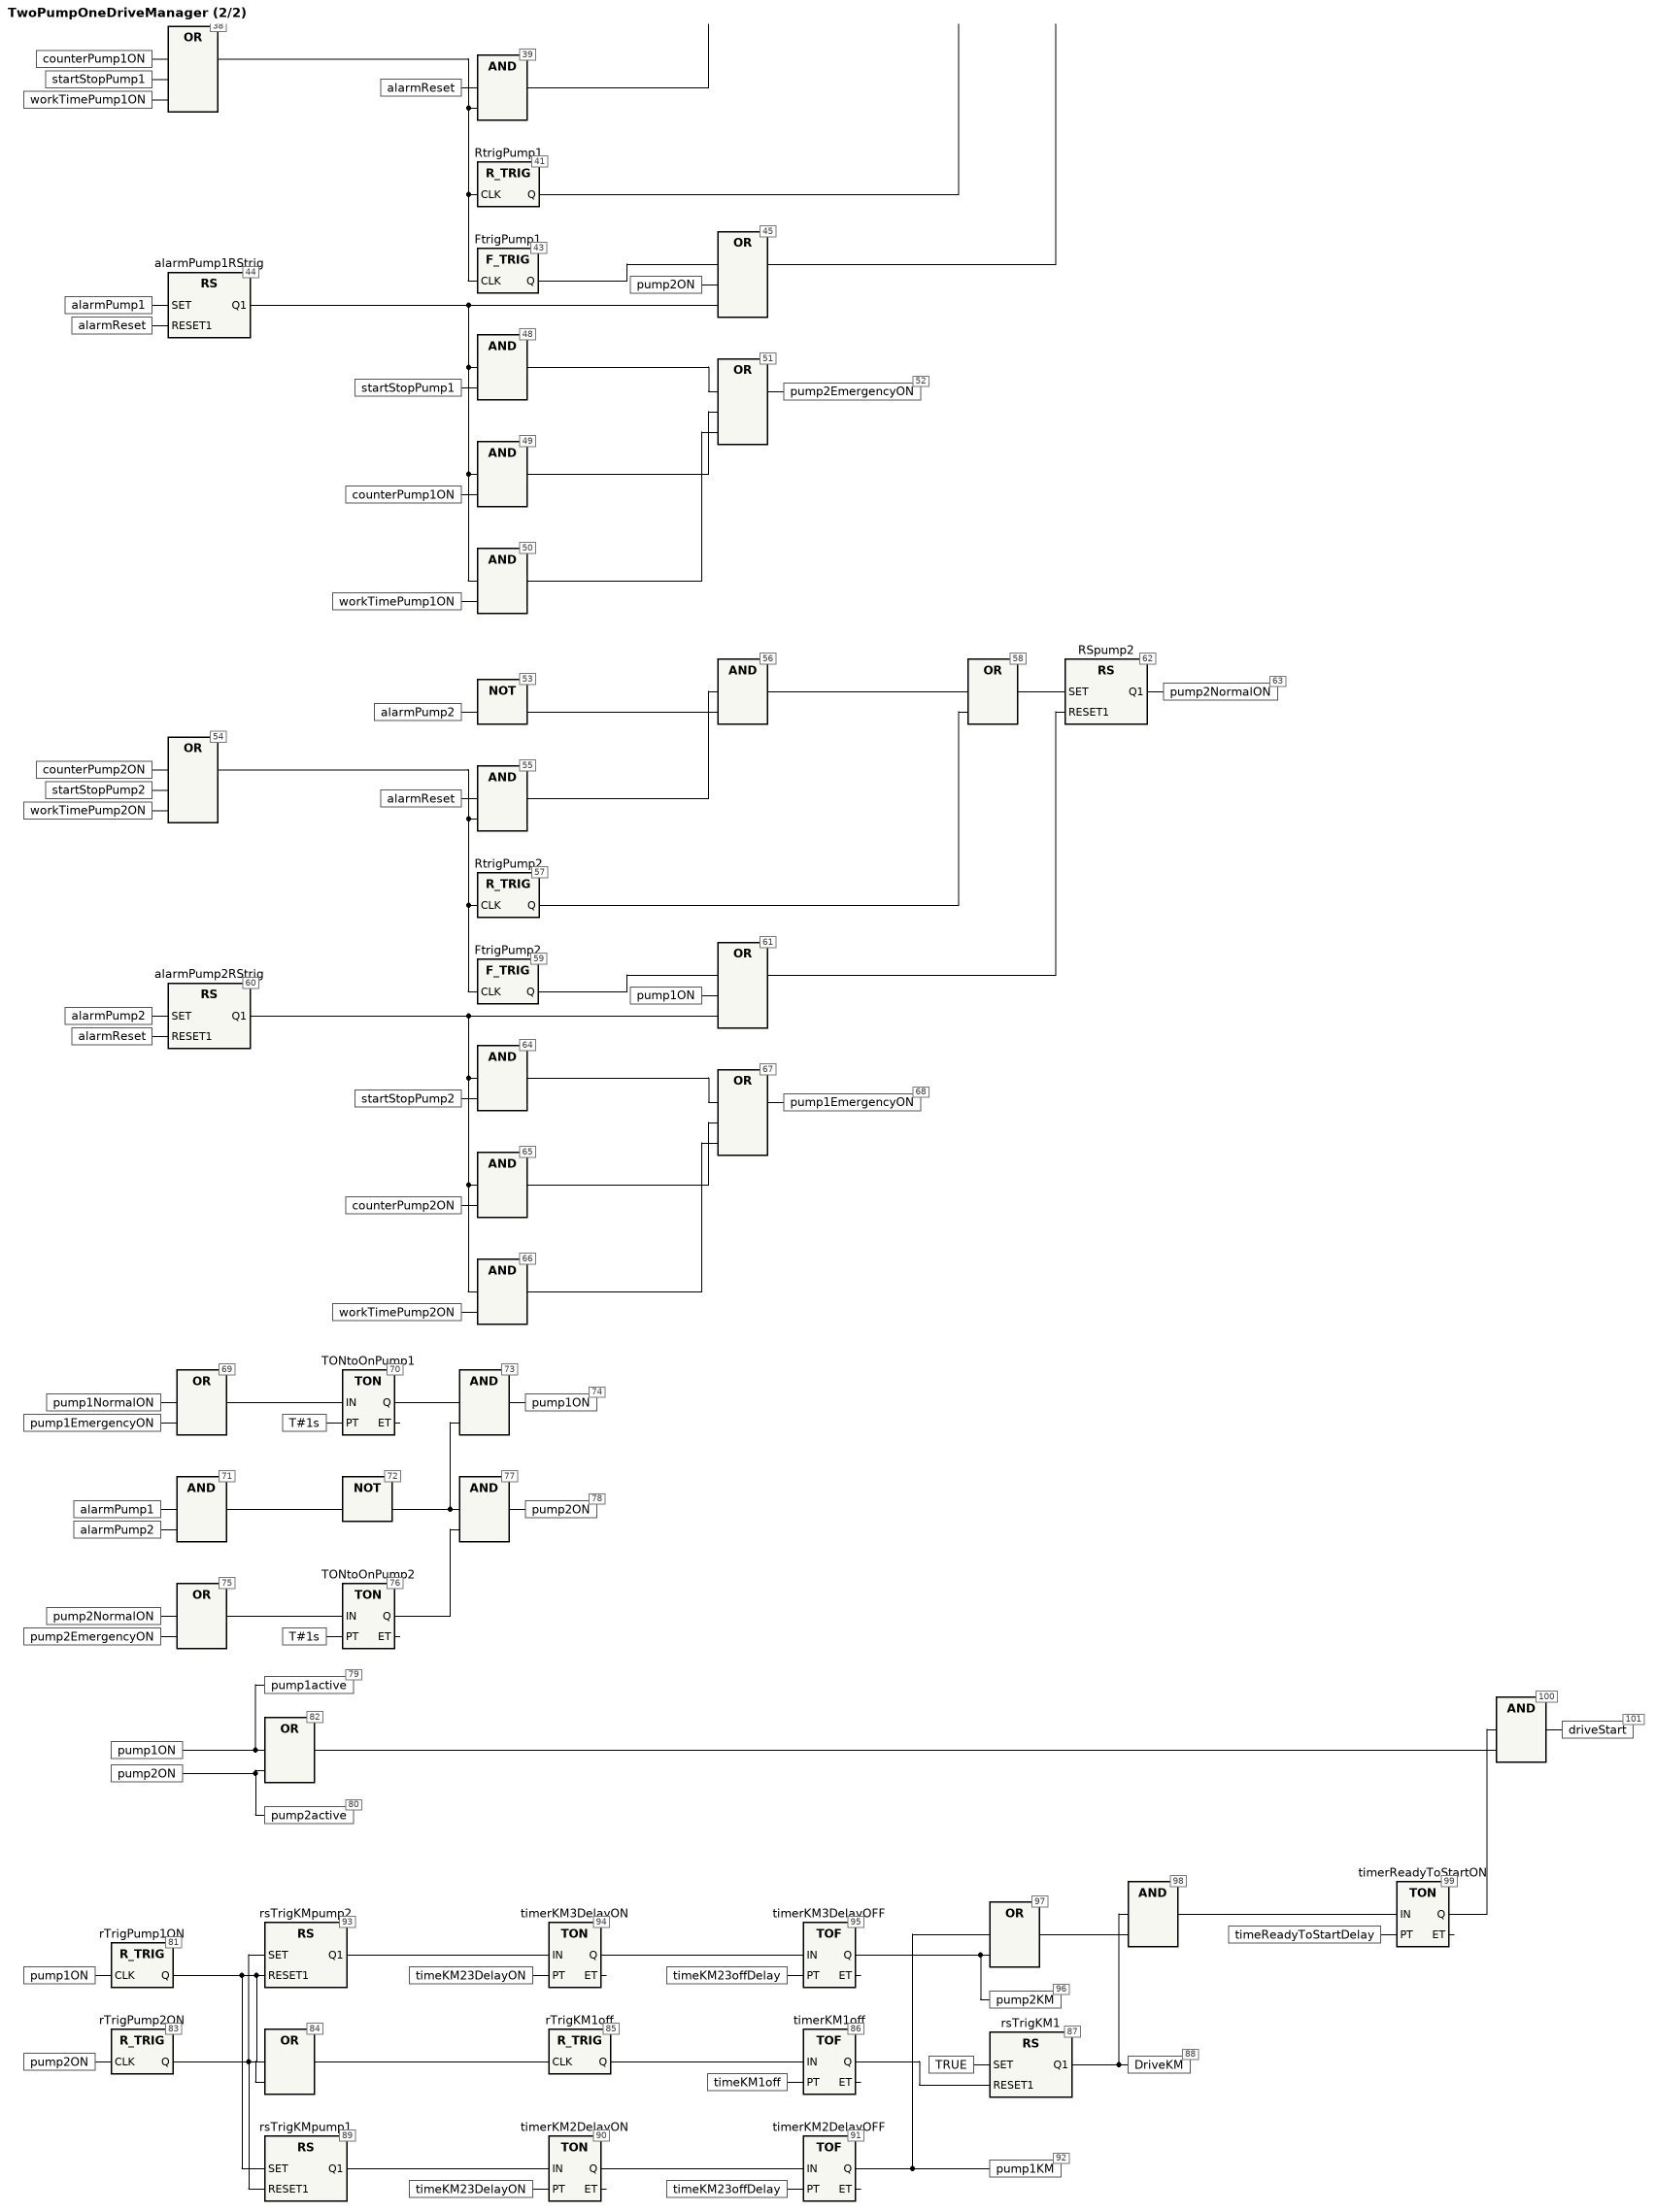
_CFC_ (* Continuous Function Chart, elements in execution order *)
(* Управление включением контактора питания ЧРП и насосов на выходе ЧРП. *)
(* Задержка на переключение. *)
(* Задержка на переключение. *)
(* Сброс времени наработки первого насоса. *)
(* Запуск насоса с наименьшей наработкой. *)
(* Блок запуска насоса с наименьшей наработкой. / Также считает наработку насосов независимо от варианта выбора запуска. *)
(* Запуск насоса с выбором по наработке. *)
(* Если workTimePump1 <= / workTimePump2, то TRUE *)
(* Если workTimePump1 > / workTimePump2, то TRUE *)
(* Счетчик времени наработки включенного насоса. *)
(* Выбор и запуск насоса с меньшим временем наработки *)
(* Текущая наработка первого насоса, сек *)
(* Блок управления запуском насосов с учетом количества включений. / При активации counterStart запустится насос с меньшим количеством включений. / При достижении счетчиком заданного значения ValueToResetCounter оба счетчика сбрасываются. *)
(* Оба счетчика сбрасываются в ноль, если хоть один достигнет заданного значения. *)
(* пуск/стоп pump2 по кол.вкл *)
(* пуск/стоп pump1 по кол.вкл *)
(* Если counterPump1 <= / counterPump2, то TRUE *)
(* выход на запуск второго насоса *)
(* запуск первого насоса при аварии второго *)
(* Если запущен первый насос, второй не включается *)
(* авария на втором насосе *)
(* ручной норм.пуск/стоп pump2 *)
(* выход на запуск первого насоса *)
(* ручной норм.пуск/стоп pump1 *)
(* запуск второго насоса при аварии первого *)
(* Если запущен второй насос, первый не включается *)
(* авария на первом насосе *)
(* Если был запущен первый насос, произошла его авария, включился второй насос, / а потом авария первого насоса ушла, сделали сброс аварии, то снова запустится первый насос. *)
(* Если был запущен второй насос, произошла его авария, включился первый насос, / а потом авария второго насоса ушла, сделали сброс аварии, то снова запустится второй насос. *)
(* Если counterPump1 > / counterPump2, то TRUE *)
(* Блок ручного управления парой насосов, которые не работают одновременно. / При аварии запущенного насоса переходит на резервный (незапущенный) насос. / Не разрешает одновременный запуск двух насосов. *)
(* пуск/стоп pump1 по наработке *)
(* пуск/стоп pump2 по наработке *)
(* Сброс времени наработки второго насоса. *)
(* КМ1, питание ЧРП *)
(* включение КМ2 (насос 1) *)
(* включение КМ3 (насос 2) *)
(* запуск ЧРП *)
(* Текущая наработка второго насоса, сек *)
#0 pulsarP1:PulsePerSec(start: Pump1ON)
#1 ADD(EN: #0.out, currentWorkTimePump1, 1)
#2 currentWorkTimePump1 <= #1
#3 pulsarP2:PulsePerSec(start: Pump2ON)
#4 ADD(EN: #3.out, currentWorkTimePump2, 1)
#5 currentWorkTimePump2 <= #4
#6 LE(currentWorkTimePump1, currentWorkTimePump2)
#7 timeStartFtrig:F_TRIG(CLK: workTimeStart)
#8 timeStartRtrig:R_TRIG(CLK: workTimeStart)
#9 AND(#6, #8.Q)
#10 RStrigTimePump1:RS(SET: #9, RESET1: #7.Q)
#11 workTimePump1ON <= #10.Q1
#12 GT(currentWorkTimePump1, currentWorkTimePump2)
#13 AND(#8.Q, #12)
#14 RStrigTimePump2:RS(SET: #13, RESET1: #7.Q)
#15 workTimePump2ON <= #14.Q1
#16 MOVE(EN: workTimePump1Reset, 0)
#17 currentWorkTimePump1 <= #16
#18 MOVE(EN: workTimePump2Reset, 0)
#19 currentWorkTimePump2 <= #18
#20 CTUPump1:CTU(CU: pump1ON, RESET: #25, PV: ValueToResetCounter)
#21 counterPump1 <= #20.CV
#22 CTUPump2:CTU(CU: pump2ON, RESET: #26, PV: ValueToResetCounter)
#23 counterPump2 <= #22.CV
#24 OR(#20.Q, #22.Q)
#25 OR(#24, Pump1ResetCounter)
#26 OR(Pump2ResetCounter, #24)
#27 LE(counterPump1, counterPump2)
#28 counterFtrig:F_TRIG(CLK: counterStart)
#29 counterRtrig:R_TRIG(CLK: counterStart)
#30 AND(#27, #29.Q)
#31 counterRStrigPump1:RS(SET: #30, RESET1: #28.Q)
#32 counterPump1ON <= #31.Q1
#33 GT(counterPump1, counterPump2)
#34 AND(#29.Q, #33)
#35 counterRStrigPump2:RS(SET: #34, RESET1: #28.Q)
#36 counterPump2ON <= #35.Q1
#37 NOT(alarmPump1)
#38 OR(counterPump1ON, startStopPump1, workTimePump1ON)
#39 AND(alarmReset, #38)
#40 AND(#39, #37)
#41 RtrigPump1:R_TRIG(CLK: #38)
#42 OR(#40, #41.Q)
#43 FtrigPump1:F_TRIG(CLK: #38)
#44 alarmPump1RStrig:RS(SET: alarmPump1, RESET1: alarmReset)
#45 OR(#43.Q, pump2ON, #44.Q1)
#46 RSpump1:RS(SET: #42, RESET1: #45)
#47 pump1NormalON <= #46.Q1
#48 AND(#44.Q1, startStopPump1)
#49 AND(#44.Q1, counterPump1ON)
#50 AND(#44.Q1, workTimePump1ON)
#51 OR(#48, #49, #50)
#52 pump2EmergencyON <= #51
#53 NOT(alarmPump2)
#54 OR(counterPump2ON, startStopPump2, workTimePump2ON)
#55 AND(alarmReset, #54)
#56 AND(#55, #53)
#57 RtrigPump2:R_TRIG(CLK: #54)
#58 OR(#56, #57.Q)
#59 FtrigPump2:F_TRIG(CLK: #54)
#60 alarmPump2RStrig:RS(SET: alarmPump2, RESET1: alarmReset)
#61 OR(#59.Q, pump1ON, #60.Q1)
#62 RSpump2:RS(SET: #58, RESET1: #61)
#63 pump2NormalON <= #62.Q1
#64 AND(#60.Q1, startStopPump2)
#65 AND(#60.Q1, counterPump2ON)
#66 AND(#60.Q1, workTimePump2ON)
#67 OR(#64, #65, #66)
#68 pump1EmergencyON <= #67
#69 OR(pump1NormalON, pump1EmergencyON)
#70 TONtoOnPump1:TON(IN: #69, PT: T#1s)
#71 AND(alarmPump1, alarmPump2)
#72 NOT(#71)
#73 AND(#70.Q, #72)
#74 pump1ON <= #73
#75 OR(pump2NormalON, pump2EmergencyON)
#76 TONtoOnPump2:TON(IN: #75, PT: T#1s)
#77 AND(#72, #76.Q)
#78 pump2ON <= #77
#79 pump1active <= pump1ON
#80 pump2active <= pump2ON
#81 rTrigPump1ON:R_TRIG(CLK: pump1ON)
#82 OR(pump1ON, pump2ON)
#83 rTrigPump2ON:R_TRIG(CLK: pump2ON)
#84 OR(#81.Q, #83.Q)
#85 rTrigKM1off:R_TRIG(CLK: #84)
#86 timerKM1off:TOF(IN: #85.Q, PT: timeKM1off)
#87 rsTrigKM1:RS(SET: TRUE, RESET1: #86.Q)
#88 DriveKM <= #87.Q1
#89 rsTrigKMpump1:RS(SET: #81.Q, RESET1: #83.Q)
#90 timerKM2DelayON:TON(IN: #89.Q1, PT: timeKM23DelayON)
#91 timerKM2DelayOFF:TOF(IN: #90.Q, PT: timeKM23offDelay)
#92 pump1KM <= #91.Q
#93 rsTrigKMpump2:RS(SET: #83.Q, RESET1: #81.Q)
#94 timerKM3DelayON:TON(IN: #93.Q1, PT: timeKM23DelayON)
#95 timerKM3DelayOFF:TOF(IN: #94.Q, PT: timeKM23offDelay)
#96 pump2KM <= #95.Q
#97 OR(#91.Q, #95.Q)
#98 AND(#87.Q1, #97)
#99 timerReadyToStartON:TON(IN: #98, PT: timeReadyToStartDelay)
#100 AND(#99.Q, #82)
#101 driveStart <= #100
_END_CFC_
END_FUNCTION_BLOCK

(* POU SimpleValve, CFC *)
FUNCTION_BLOCK SimpleValve
VAR_INPUT
	inputOpen: BOOL;		(*вход подающий сигнал на открытие*)
	inputClose: BOOL;		(*вход, подающий сигнал на закрытие*)
	statusOpen: BOOL;		(*статус: заслонка/задвижка ОТКРЫТА*)
	statusClose: BOOL;		(*статус: заслонка/задвижка ЗАКРЫТА*)
	reset: BOOL;		(*ручной сброс выходов и аварий в неактивное состояние*)
	timeToOpenClose: TIME;		(*Время в секундах на открытие/закрытие (по тех.характеристикам прибора).*)
END_VAR
VAR_OUTPUT
	outputOpen: BOOL;		(*выход на открытие задвижки/заслонки*)
	outputClose: BOOL;		(*выход на закрытие задвижки/заслонки*)
	errorToOpen: BOOL;		(*авария на открытие - задвижка не открылась за заданное время.*)
	errorToClose: BOOL;		(*авария на закрытие - задвижка не закрылась за заданное время.*)
END_VAR
VAR
	toOpenTrigger: RS;
	toCloseTrigger: RS;
	timerToOpenClose: TON;
	timerToDelayOPen: TOF;
	timerToDelayClose: TOF;
	timerToStopOpening: TOF;
	timerToStopClosing: TOF;
END_VAR
VAR (* helpers for the ST form of the networks *)
	_t25 : BOOL;
	_t26 : BOOL;
	_t22 : BOOL;
	_t23 : BOOL;
END_VAR
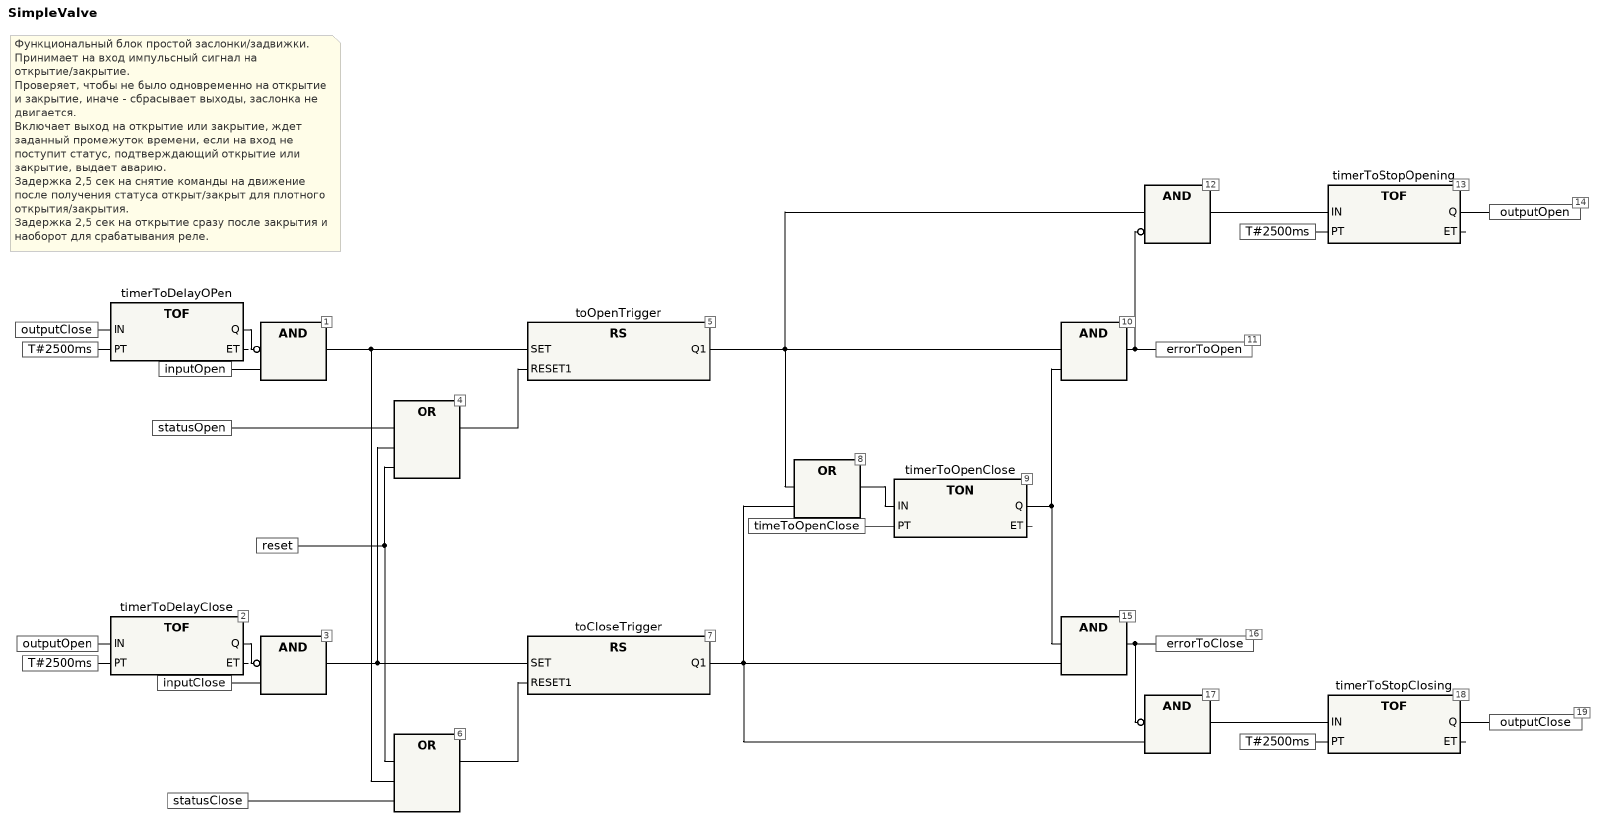
_CFC_ (* Continuous Function Chart, elements in execution order *)
(* Функциональный блок простой заслонки/задвижки. / Принимает на вход импульсный сигнал на открытие/закрытие. / Проверяет, чтобы не было одновременно на открытие и закрытие, иначе - сбрасывает выходы, заслонка не двигается. / Включает выход на открытие или закрытие, ждет заданный промежуток времени, если на вход не поступит статус, подтверждающий открытие или закрытие, выдает аварию. / Задержка 2,5 сек на снятие команды на движение после получения статуса открыт/закрыт для плотного открытия/закрытия. / Задержка 2,5 сек на открытие сразу после закрытия и наоборот для срабатывания реле. *)
#0 timerToDelayOPen:TOF(IN: outputClose, PT: T#2500ms)
#1 AND(NOT #0.Q, inputOpen)
#2 timerToDelayClose:TOF(IN: outputOpen, PT: T#2500ms)
#3 AND(NOT #2.Q, inputClose)
#4 OR(statusOpen, #3, reset)
#5 toOpenTrigger:RS(SET: #1, RESET1: #4)
#6 OR(reset, #1, statusClose)
#7 toCloseTrigger:RS(SET: #3, RESET1: #6)
#8 OR(#5.Q1, #7.Q1)
#9 timerToOpenClose:TON(IN: #8, PT: timeToOpenClose)
#10 AND(#5.Q1, #9.Q)
#11 errorToOpen <= #10
#12 AND(#5.Q1, NOT #10)
#13 timerToStopOpening:TOF(IN: #12, PT: T#2500ms)
#14 outputOpen <= #13.Q
#15 AND(#9.Q, #7.Q1)
#16 errorToClose <= #15
#17 AND(NOT #15, #7.Q1)
#18 timerToStopClosing:TOF(IN: #17, PT: T#2500ms)
#19 outputClose <= #18.Q
_END_CFC_
(* the same logic as Structured Text *)
(* Функциональный блок простой заслонки/задвижки. / Принимает на вход импульсный сигнал на открытие/закрытие. / Проверяет, чтобы не было одновременно на открытие и закрытие, иначе - сбрасывает выходы, заслонка не двигается. / Включает выход на открытие или закрытие, ждет заданный промежуток времени, если на вход не поступит статус, подтверждающий открытие или закрытие, выдает аварию. / Задержка 2,5 сек на снятие команды на движение после получения статуса открыт/закрыт для плотного открытия/закрытия. / Задержка 2,5 сек на открытие сразу после закрытия и наоборот для срабатывания реле. *)
timerToDelayOPen(IN := outputClose, PT := T#2500ms);
_t25 := NOT timerToDelayOPen.Q AND inputOpen;
timerToDelayClose(IN := outputOpen, PT := T#2500ms);
_t26 := NOT timerToDelayClose.Q AND inputClose;
toOpenTrigger(SET := _t25, RESET1 := statusOpen OR _t26 OR reset);
toCloseTrigger(SET := _t26, RESET1 := reset OR _t25 OR statusClose);
timerToOpenClose(IN := toOpenTrigger.Q1 OR toCloseTrigger.Q1, PT := timeToOpenClose);
_t22 := toOpenTrigger.Q1 AND timerToOpenClose.Q;
errorToOpen := _t22;
timerToStopOpening(IN := toOpenTrigger.Q1 AND NOT _t22, PT := T#2500ms);
outputOpen := timerToStopOpening.Q;
_t23 := timerToOpenClose.Q AND toCloseTrigger.Q1;
errorToClose := _t23;
timerToStopClosing(IN := NOT _t23 AND toCloseTrigger.Q1, PT := T#2500ms);
outputClose := timerToStopClosing.Q;
END_FUNCTION_BLOCK

(* POU FilterQueueManager, CFC *)
FUNCTION_BLOCK FilterQueueManager
VAR_INPUT
	input: BOOL;		(*Вход на старт регенерации.*)
	filterAlarm: BOOL;		(*Вход аварии от управляющего клапана фильтра.*)
	regenFilterStatus: BOOL;		(*Вход для сигнала подтверждения начала регенерации
			от фильтра.*)
	alarmReset: BOOL;		(*Сброс статуса о неудачной попытке регенерации.*)
	startNextLoop: BOOL;		(*Сбрасывает сигнал о том, что регенерация уже была.
			Применять для начала нового цикла.*)
END_VAR
VAR_OUTPUT
	output: BOOL;		(*Выход, передающий сигнал от счетчика о начале регенерации,
			на следующий фильтр. Соединять с input.*)
	regenFilterOUT: BOOL;		(*Выход на старт регенерации, подаваемый на фильтр.*)
	regenerated: BOOL;		(*TRUE, если этот фильтр уже промыт.*)
	failToRegen: BOOL;		(*Не удалось запустить регенерацию.
			Не пришло подтверждение от фильтра более 5 сек после старта.*)
	counterReset: BOOL;		(*Сбросить счетчик начала регенерации для отсчета следующего.
			Подключать только от первого фильтр в цепи.*)
	regenFinished: BOOL;		(*Импульсный сигнал, возникающий при отключени сигнала подтверждения
			статуса промывки от фильтра (фильтр вернулся в режим фильтрации) или при неудачной попытке регенерации. 
			Использовать для старта нового цикла.*)
END_VAR
VAR
	regStatusDelay: TON;		(*Таймер задержки ожидания подтверждения от фильтра
			о начале регенерации.*)
	regStartRS: RS;		(*Триггер старта регенерации.*)
	failureRS: RS;		(*Триггер неудачного пуска регенерации.*)
	successRS: RS;		(*Триггер удачной регенерации.*)
	counterResetRtrig: R_TRIG;		(*Детектор переднего фронта на сброс счетчика.*)
	regenFilterOFF: F_TRIG;		(*Триггер контроля отключения сигнала от фильтра, что он закончил
			режим промывки для возврата задвижек обратно в режим фильтрации.*)
	failureRtrig: R_TRIG;		(*детектор переднего фронта сигнала о неудачной попытке регенерации.*)
END_VAR
VAR (* helpers for the ST form of the networks *)
	_t45 : BOOL;
	_t78 : BOOL;
END_VAR
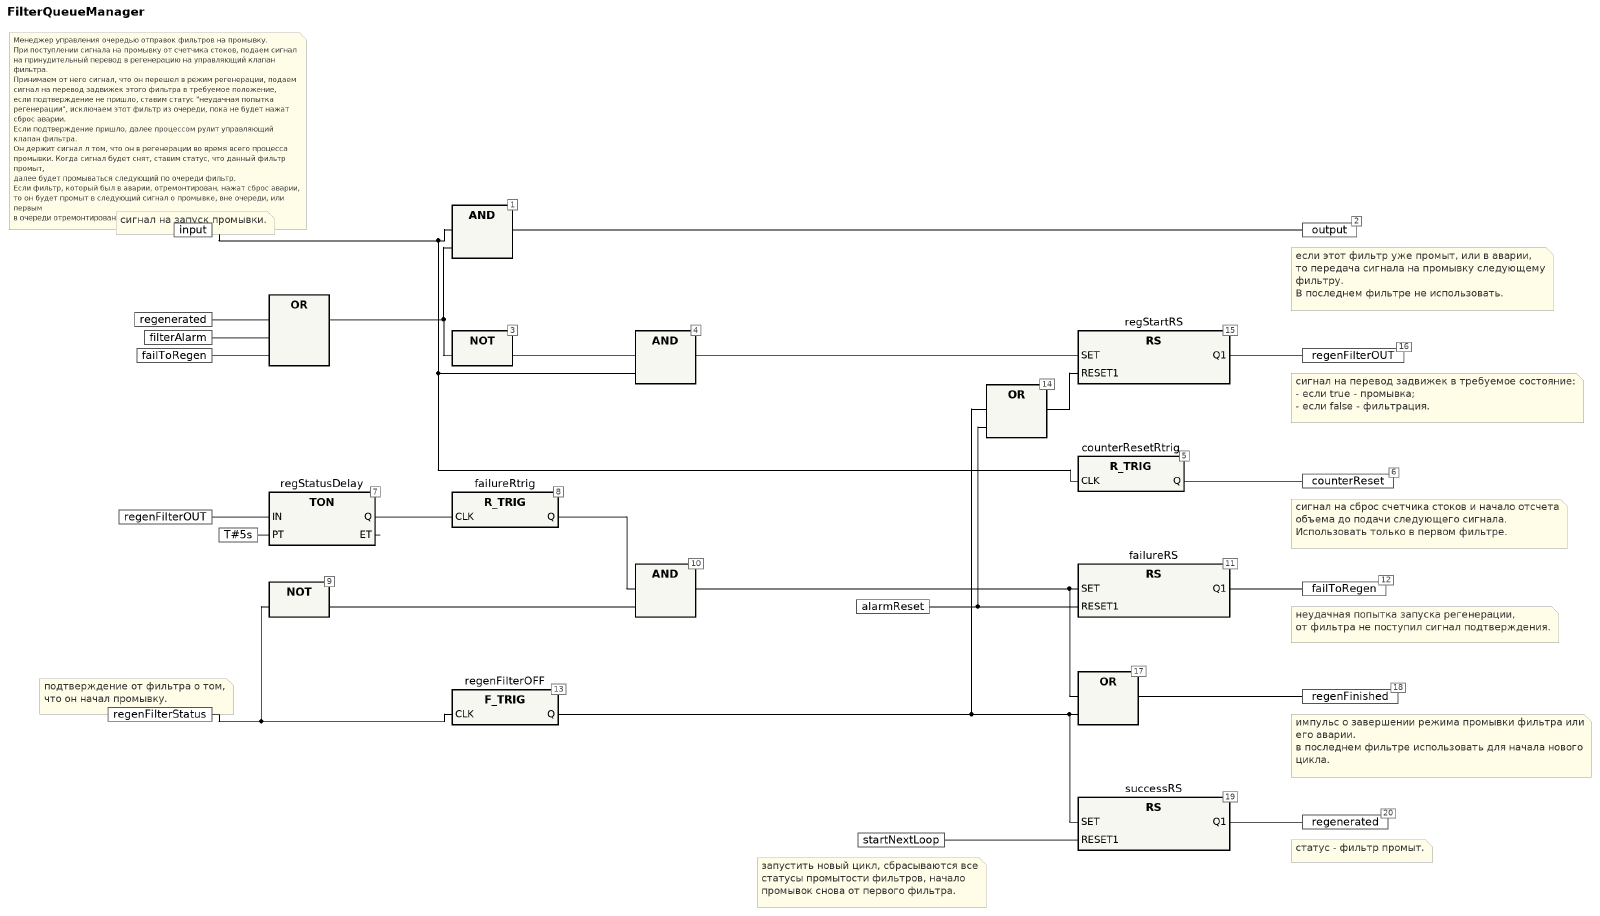
_CFC_ (* Continuous Function Chart, elements in execution order *)
(* запустить новый цикл, сбрасываются все / статусы промытости фильтров, начало / промывок снова от первого фильтра. *)
(* Менеджер управления очередью отправок фильтров на промывку. / При поступлении сигнала на промывку от счетчика стоков, подаем сигнал на принудительный перевод в регенерацию на управляющий клапан фильтра. / Принимаем от него сигнал, что он перешел в режим регенерации, подаем сигнал на перевод задвижек этого фильтра в требуемое положение, / если подтверждение не пришло, ставим статус "неудачная попытка регенерации", исключаем этот фильтр из очереди, пока не будет нажат сброс аварии. / Если подтверждение пришло, далее процессом рулит управляющий клапан фильтра. / Он держит сигнал л том, что он в регенерации во время всего процесса промывки. Когда сигнал будет снят, ставим статус, что данный фильтр промыт, / далее будет промываться следующий по очереди фильтр. / Если фильтр, который был в аварии, отремонтирован, нажат сброс аварии, то он будет промыт в следующий сигнал о промывке, вне очереди, или первым / в очереди отремонтированных, после чего пойдет обычная очередь. *)
(* сигнал на запуск промывки. *)
(* если этот фильтр уже промыт, или в аварии, / то передача сигнала на промывку следующему фильтру. / В последнем фильтре не использовать. *)
(* сигнал на перевод задвижек в требуемое состояние: / - если true - промывка; / - если false - фильтрация. *)
(* сигнал на сброс счетчика стоков и начало отсчета / объема до подачи следующего сигнала. / Использовать только в первом фильтре. *)
(* неудачная попытка запуска регенерации, / от фильтра не поступил сигнал подтверждения. *)
(* статус - фильтр промыт. *)
(* подтверждение от фильтра о том, / что он начал промывку. *)
(* импульс о завершении режима промывки фильтра или его аварии. / в последнем фильтре использовать для начала нового цикла. *)
#0 OR(regenerated, filterAlarm, failToRegen)
#1 AND(input, #0)
#2 output <= #1
#3 NOT(#0)
#4 AND(#3, input)
#5 counterResetRtrig:R_TRIG(CLK: input)
#6 counterReset <= #5.Q
#7 regStatusDelay:TON(IN: regenFilterOUT, PT: T#5s)
#8 failureRtrig:R_TRIG(CLK: #7.Q)
#9 NOT(regenFilterStatus)
#10 AND(#8.Q, #9)
#11 failureRS:RS(SET: #10, RESET1: alarmReset)
#12 failToRegen <= #11.Q1
#13 regenFilterOFF:F_TRIG(CLK: regenFilterStatus)
#14 OR(#13.Q, alarmReset)
#15 regStartRS:RS(SET: #4, RESET1: #14)
#16 regenFilterOUT <= #15.Q1
#17 OR(#10, #13.Q)
#18 regenFinished <= #17
#19 successRS:RS(SET: #13.Q, RESET1: startNextLoop)
#20 regenerated <= #19.Q1
_END_CFC_
(* the same logic as Structured Text *)
(* запустить новый цикл, сбрасываются все / статусы промытости фильтров, начало / промывок снова от первого фильтра. *)
(* Менеджер управления очередью отправок фильтров на промывку. / При поступлении сигнала на промывку от счетчика стоков, подаем сигнал на принудительный перевод в регенерацию на управляющий клапан фильтра. / Принимаем от него сигнал, что он перешел в режим регенерации, подаем сигнал на перевод задвижек этого фильтра в требуемое положение, / если подтверждение не пришло, ставим статус "неудачная попытка регенерации", исключаем этот фильтр из очереди, пока не будет нажат сброс аварии. / Если подтверждение пришло, далее процессом рулит управляющий клапан фильтра. / Он держит сигнал л том, что он в регенерации во время всего процесса промывки. Когда сигнал будет снят, ставим статус, что данный фильтр промыт, / далее будет промываться следующий по очереди фильтр. / Если фильтр, который был в аварии, отремонтирован, нажат сброс аварии, то он будет промыт в следующий сигнал о промывке, вне очереди, или первым / в очереди отремонтированных, после чего пойдет обычная очередь. *)
(* сигнал на запуск промывки. *)
(* если этот фильтр уже промыт, или в аварии, / то передача сигнала на промывку следующему фильтру. / В последнем фильтре не использовать. *)
(* сигнал на перевод задвижек в требуемое состояние: / - если true - промывка; / - если false - фильтрация. *)
(* сигнал на сброс счетчика стоков и начало отсчета / объема до подачи следующего сигнала. / Использовать только в первом фильтре. *)
(* неудачная попытка запуска регенерации, / от фильтра не поступил сигнал подтверждения. *)
(* статус - фильтр промыт. *)
(* подтверждение от фильтра о том, / что он начал промывку. *)
(* импульс о завершении режима промывки фильтра или его аварии. / в последнем фильтре использовать для начала нового цикла. *)
_t45 := regenerated OR filterAlarm OR failToRegen;
output := input AND _t45;
counterResetRtrig(CLK := input);
counterReset := counterResetRtrig.Q;
regStatusDelay(IN := regenFilterOUT, PT := T#5s);
failureRtrig(CLK := regStatusDelay.Q);
_t78 := failureRtrig.Q AND NOT regenFilterStatus;
failureRS(SET := _t78, RESET1 := alarmReset);
failToRegen := failureRS.Q1;
regenFilterOFF(CLK := regenFilterStatus);
regStartRS(SET := NOT _t45 AND input, RESET1 := regenFilterOFF.Q OR alarmReset);
regenFilterOUT := regStartRS.Q1;
regenFinished := _t78 OR regenFilterOFF.Q;
successRS(SET := regenFilterOFF.Q, RESET1 := startNextLoop);
regenerated := successRS.Q1;
END_FUNCTION_BLOCK

(* POU TimeFromWorkTime, ST *)
FUNCTION_BLOCK TimeFromWorkTime
VAR_INPUT
	 input: DWORD; (*Вход счетчика от счетчика наработки, сек.*)
END_VAR
VAR_OUTPUT
	days: WORD; (*Выход наработка, дней*)
	hours: WORD; (*Выход наработка, часов*)
	minutes: WORD; (*Выход наработка, минут*)
	seconds: WORD; (*Выход наработка, секунд*)
END_VAR
VAR
	temp: DWORD;
END_VAR
days:= DWORD_TO_WORD (input / (60 * 60 * 24));
temp:= input MOD (60 * 60 * 24);
hours:= DWORD_TO_WORD (temp / (60 * 60));
temp:= temp MOD (60 * 60);
minutes:= DWORD_TO_WORD (temp / 60);
temp:= temp MOD 60;
seconds:= DWORD_TO_WORD (temp);
END_FUNCTION_BLOCK

(* POU CounterTwoPumpManager, CFC *)
FUNCTION_BLOCK CounterTwoPumpManager
VAR_INPUT
	startStopPump1: BOOL;		(*Сигнал на пуск/стоп первого насоса.*)
	startStopPump2: BOOL;		(*Сигнал на пуск/стоп второго насоса.*)
	alarmPump1: BOOL;		(*Сигнал "авария" на первом насосе.*)
	alarmPump2: BOOL;		(*Сигнал "авария" на втором насосе.*)
	alarmReset: BOOL;		(*Сброс аварии.*)

	counterStart: BOOL;		(*Запуск насоса с меньшим количеством включений.*)
	Pump1ResetCounter: BOOL;		(*Сброс счетчика количества включений первого насоса. Сбрасывается также автоматически при достижении счетчиком значения ValueToResetCTU.*)
	Pump2ResetCounter: BOOL;		(*Сброс счетчика количества включений второго насоса. Сбрасывается также автоматически при достижении счетчиком значения ValueToResetCTU.*)
	ValueToResetCounter: WORD := 32767;		(*Значение счетчика, после которого он сбрасывается на ноль.
			Максимальное допустимое значение: 32767, будет установлено, если не подключать ничего на вход.*)
END_VAR
VAR_OUTPUT
	pump1ON: BOOL;		(*Выход на включение первого насоса.*)
	pump2ON: BOOL;		(*Выход на включение второго насоса.*)

	counterPump1: WORD;		(*Количество включений первого насоса. При достижении значения ValueToResetCTU сбрасывается в ноль.*)
	counterPump2: WORD;		(*Количество включений второго насоса. При достижении значения ValueToResetCTU сбрасывается в ноль.*)
END_VAR
VAR
	RtrigPump1: R_TRIG;		(*Включает первый насос по фронту сигнала на ручной пуск/стоп.*)
	FtrigPump1: F_TRIG;		(*Выключает первый насос по спаду сигнала на ручной пуск/стоп.*)
	RtrigPump2: R_TRIG;		(*Включает второй насос по фронту сигнала на ручной пуск/стоп.*)
	FtrigPump2: F_TRIG;		(*Выключает второй насос по спаду сигнала на ручной пуск/стоп.*)
	RSpump1: RS;		(*RS-триггер нормального включения первого насоса*)
	RSpump2: RS;		(*RS-триггер нормального включения второго насоса*)
	pump1NormalON: BOOL;		(*Сигнал нормального (неаварийного) включения первого насоса.*)
	pump2NormalON: BOOL;		(*Сигнал нормального (неаварийного) включения второго насоса.*)
	pump2EmergencyON: BOOL;		(*Сигнал аварийного включения второго насоса (при аварии первого).*)
	pump1EmergencyON: BOOL;		(*Сигнал аварийного включения первого насоса (при аварии второго).*)
	alarmPump1RStrig: RS;		(*Триггер аварии первого насоса.*)
	alarmPump2RStrig: RS;		(*Триггер аварии второго насоса.*)
	TONtoOnPump1: TON;		(*Таймер задержки включения первого насоса, на переключение контакторов при аварийном переключении.
			Жестко задано 1 секунда.*)
	TONtoOnPump2: TON;		(*Таймер задержки включения второго насоса, на переключение контакторов при аварийном переключении.
						Жестко задано 1 секунда.*)

	CTUPump1: CTU;		(*Счетчик количества включений первого насоса.*)
	CTUPump2: CTU;		(*Счетчик количества включений второго насоса.*)
	counterRtrig: R_TRIG;		(*Детектор переднего фронта сигнала на старт насоса с меньшей наработкой, включает насос.*)
	counterFtrig: F_TRIG;		(*Детектор спада сигнала на запуск насоса с меньшей наработкой, останавливает насос.*)
	counterRStrigPump1: RS;		(*Триггер-защелка включения первого насоса при запуске по количеству включений.*)
	counterRStrigPump2: RS;		(*Триггер-защелка включения второго насоса при запуске по количеству включений.*)
	counterPump1ON: BOOL;		(*Сигнал на запуск первого насоса при запуске по количеству включений.*)
	counterPump2ON: BOOL;		(*Сигнал на запуск второго насоса при запуске по количеству включений.*)

END_VAR
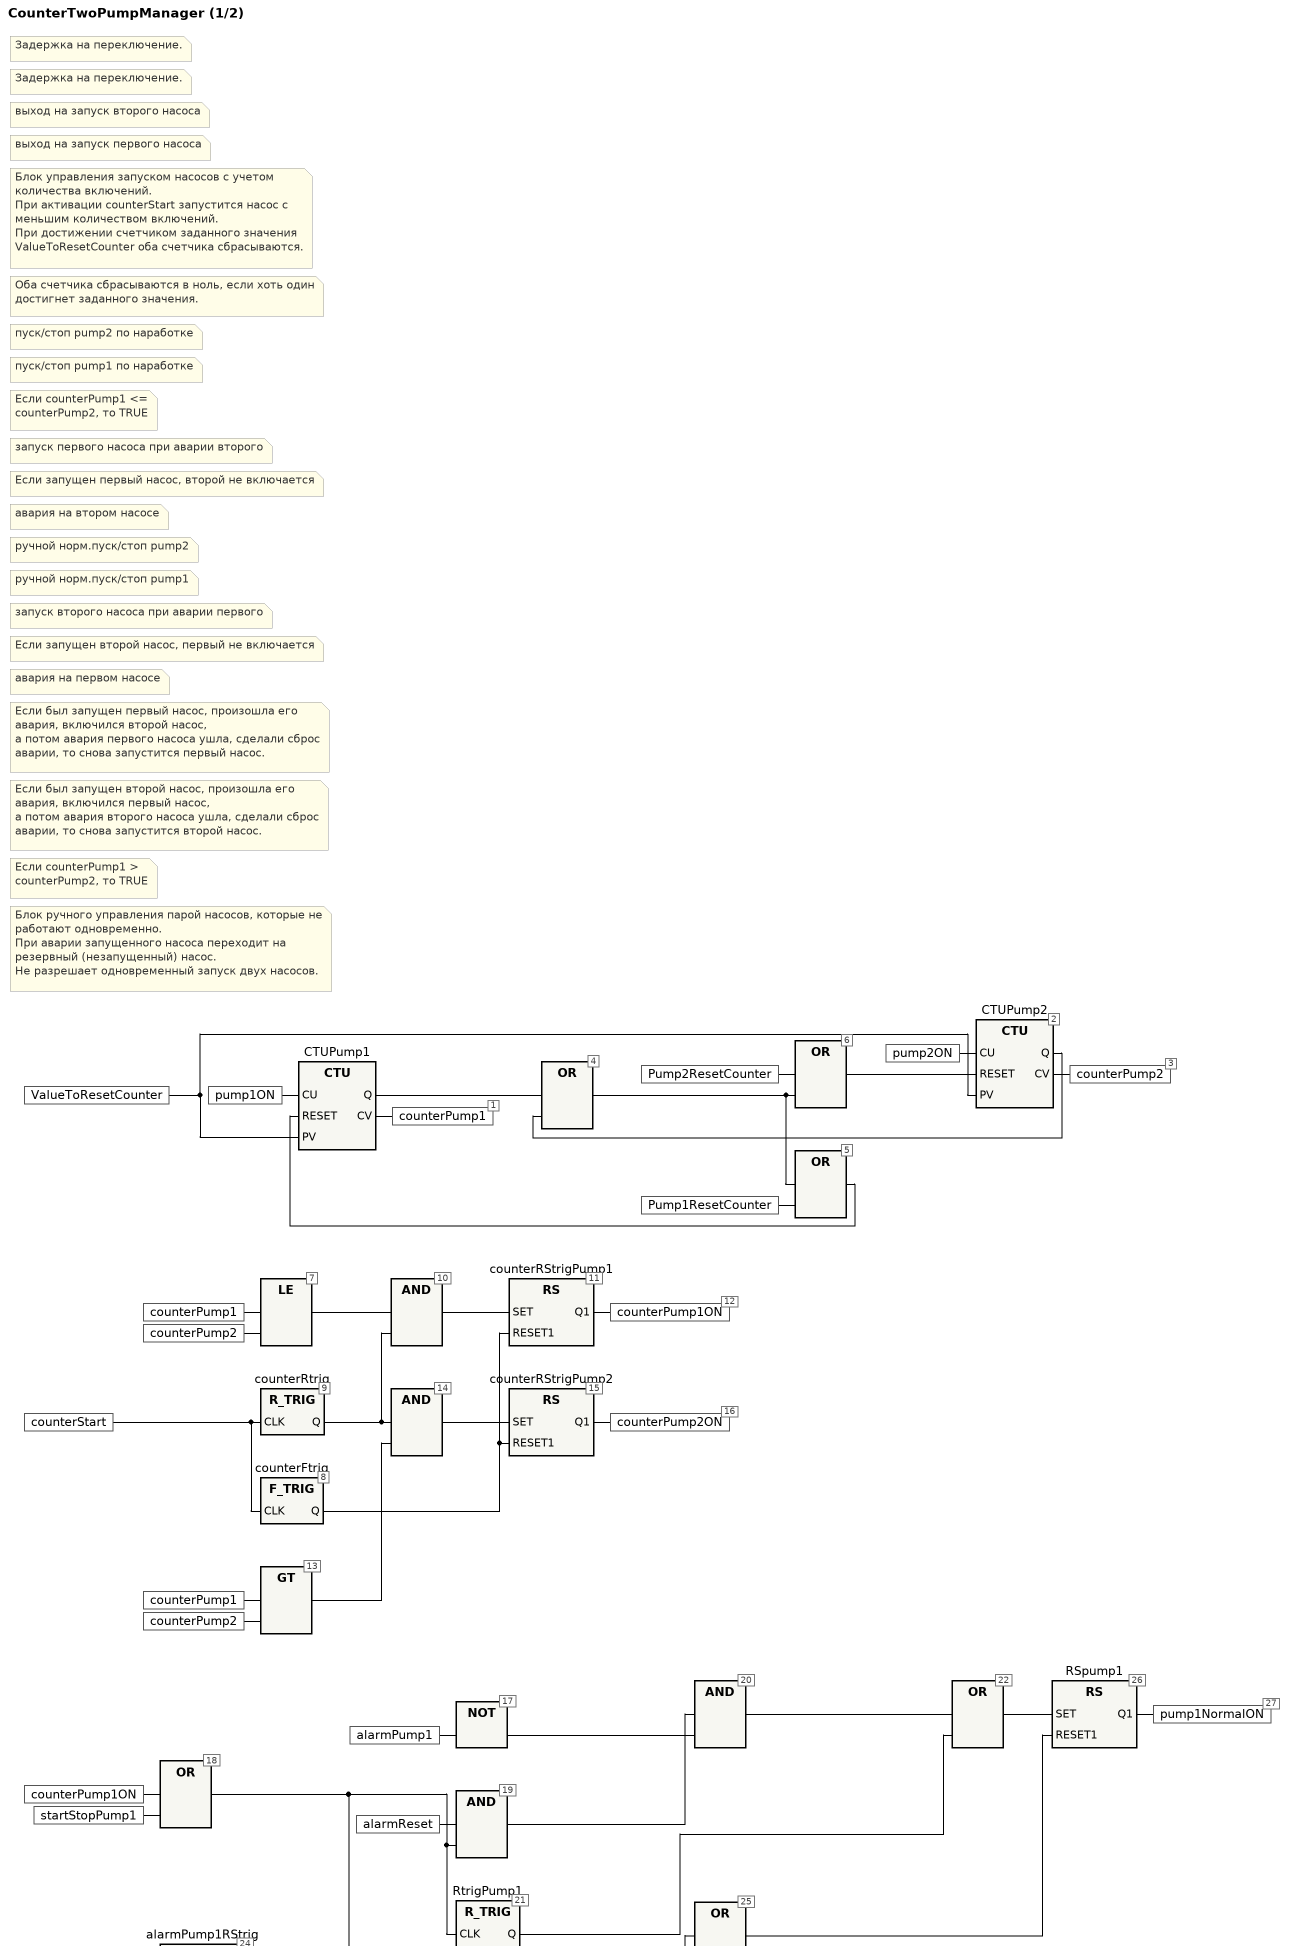
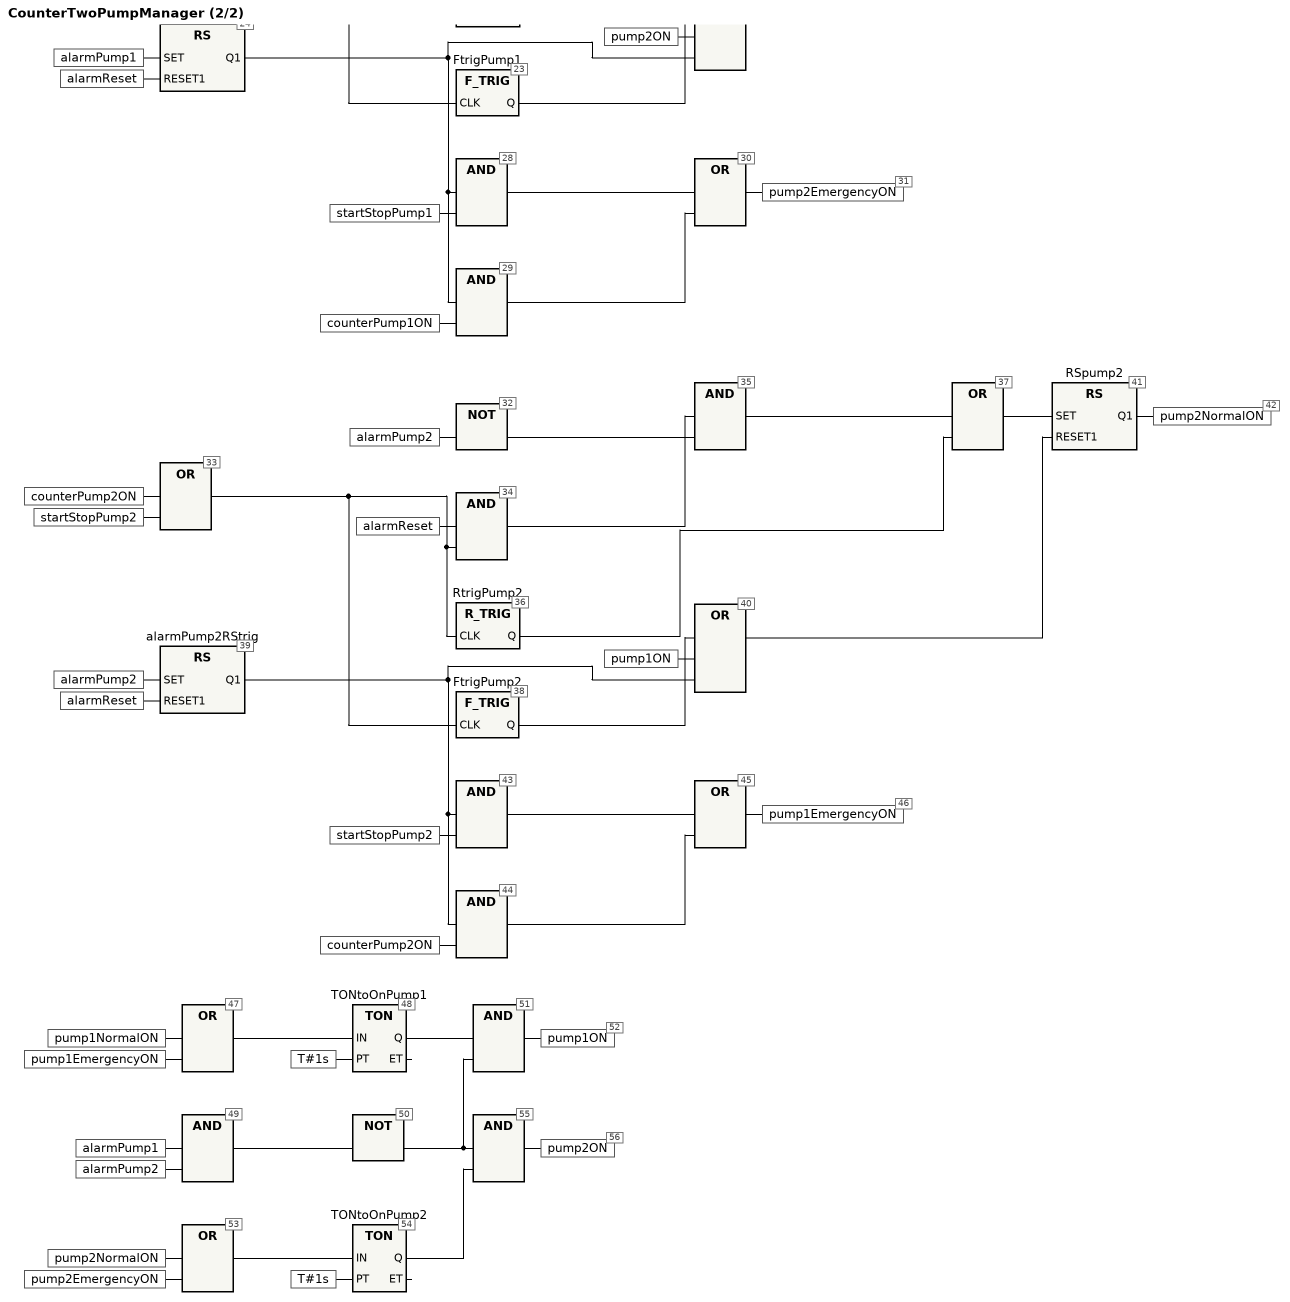
_CFC_ (* Continuous Function Chart, elements in execution order *)
(* Задержка на переключение. *)
(* Задержка на переключение. *)
(* выход на запуск второго насоса *)
(* выход на запуск первого насоса *)
(* Блок управления запуском насосов с учетом количества включений. / При активации counterStart запустится насос с меньшим количеством включений. / При достижении счетчиком заданного значения ValueToResetCounter оба счетчика сбрасываются. *)
(* Оба счетчика сбрасываются в ноль, если хоть один достигнет заданного значения. *)
(* пуск/стоп pump2 по наработке *)
(* пуск/стоп pump1 по наработке *)
(* Если counterPump1 <= / counterPump2, то TRUE *)
(* запуск первого насоса при аварии второго *)
(* Если запущен первый насос, второй не включается *)
(* авария на втором насосе *)
(* ручной норм.пуск/стоп pump2 *)
(* ручной норм.пуск/стоп pump1 *)
(* запуск второго насоса при аварии первого *)
(* Если запущен второй насос, первый не включается *)
(* авария на первом насосе *)
(* Если был запущен первый насос, произошла его авария, включился второй насос, / а потом авария первого насоса ушла, сделали сброс аварии, то снова запустится первый насос. *)
(* Если был запущен второй насос, произошла его авария, включился первый насос, / а потом авария второго насоса ушла, сделали сброс аварии, то снова запустится второй насос. *)
(* Если counterPump1 > / counterPump2, то TRUE *)
(* Блок ручного управления парой насосов, которые не работают одновременно. / При аварии запущенного насоса переходит на резервный (незапущенный) насос. / Не разрешает одновременный запуск двух насосов. *)
#0 CTUPump1:CTU(CU: pump1ON, RESET: #5, PV: ValueToResetCounter)
#1 counterPump1 <= #0.CV
#2 CTUPump2:CTU(CU: pump2ON, RESET: #6, PV: ValueToResetCounter)
#3 counterPump2 <= #2.CV
#4 OR(#0.Q, #2.Q)
#5 OR(#4, Pump1ResetCounter)
#6 OR(Pump2ResetCounter, #4)
#7 LE(counterPump1, counterPump2)
#8 counterFtrig:F_TRIG(CLK: counterStart)
#9 counterRtrig:R_TRIG(CLK: counterStart)
#10 AND(#7, #9.Q)
#11 counterRStrigPump1:RS(SET: #10, RESET1: #8.Q)
#12 counterPump1ON <= #11.Q1
#13 GT(counterPump1, counterPump2)
#14 AND(#9.Q, #13)
#15 counterRStrigPump2:RS(SET: #14, RESET1: #8.Q)
#16 counterPump2ON <= #15.Q1
#17 NOT(alarmPump1)
#18 OR(counterPump1ON, startStopPump1)
#19 AND(alarmReset, #18)
#20 AND(#19, #17)
#21 RtrigPump1:R_TRIG(CLK: #18)
#22 OR(#20, #21.Q)
#23 FtrigPump1:F_TRIG(CLK: #18)
#24 alarmPump1RStrig:RS(SET: alarmPump1, RESET1: alarmReset)
#25 OR(#23.Q, pump2ON, #24.Q1)
#26 RSpump1:RS(SET: #22, RESET1: #25)
#27 pump1NormalON <= #26.Q1
#28 AND(#24.Q1, startStopPump1)
#29 AND(#24.Q1, counterPump1ON)
#30 OR(#28, #29)
#31 pump2EmergencyON <= #30
#32 NOT(alarmPump2)
#33 OR(counterPump2ON, startStopPump2)
#34 AND(alarmReset, #33)
#35 AND(#34, #32)
#36 RtrigPump2:R_TRIG(CLK: #33)
#37 OR(#35, #36.Q)
#38 FtrigPump2:F_TRIG(CLK: #33)
#39 alarmPump2RStrig:RS(SET: alarmPump2, RESET1: alarmReset)
#40 OR(#38.Q, pump1ON, #39.Q1)
#41 RSpump2:RS(SET: #37, RESET1: #40)
#42 pump2NormalON <= #41.Q1
#43 AND(#39.Q1, startStopPump2)
#44 AND(#39.Q1, counterPump2ON)
#45 OR(#43, #44)
#46 pump1EmergencyON <= #45
#47 OR(pump1NormalON, pump1EmergencyON)
#48 TONtoOnPump1:TON(IN: #47, PT: T#1s)
#49 AND(alarmPump1, alarmPump2)
#50 NOT(#49)
#51 AND(#48.Q, #50)
#52 pump1ON <= #51
#53 OR(pump2NormalON, pump2EmergencyON)
#54 TONtoOnPump2:TON(IN: #53, PT: T#1s)
#55 AND(#50, #54.Q)
#56 pump2ON <= #55
_END_CFC_
END_FUNCTION_BLOCK

(* POU ImpulsCounter, CFC *)
FUNCTION_BLOCK ImpulsCounter
VAR_INPUT
	impulsInput: BOOL;		(*ходящие импульсы от расходомера.
			Каждый импульс будет прибавлять в итоговую сумму величину веса импульса.*)
	impulsValue: REAL;		(*Вес импульса расходомера.*)
	resetCounter: BOOL;		(*Сброс счетчика.*)
	correctionValue: REAL;		(*Число, которое будет прибавлено или вычтено из накопленной суммы.*)
	addCorrection: BOOL;		(*Прибавить коррекцию к накопленной сумме.*)
	deleteCorrection: BOOL;		(*Вычесть коррекцию из накопленной суммы.
			Если получится отрицательное число, сумма скинется в ноль.*)
END_VAR
VAR_OUTPUT
	totalAmountREAL: REAL;		(*Накопленная сумма в рациональном виде.
			В какой-то момент может выводится в экспоненциальной форме.*)
	totalAmountUDINT: UDINT;		(*Накопленная сумма в целочисленном виде.
			Округление десятичных по правилам арифметики.*)
END_VAR
VAR
	inputImpulsRtrig: R_TRIG;		(*Детектор переднего фронта входящих импульсов.*)
	resetRtrig: R_TRIG;		(*Детектор переднего фронта сигнала на сброс счетчика.*)
	addCorrRtrig: R_TRIG;		(*Детектор переднего фронта сигнала на прибавление коррекции.*)
	deleteCorrRtrig: R_TRIG;		(*Детектор переднего фронта сигнала на вычитание коррекции.*)
END_VAR
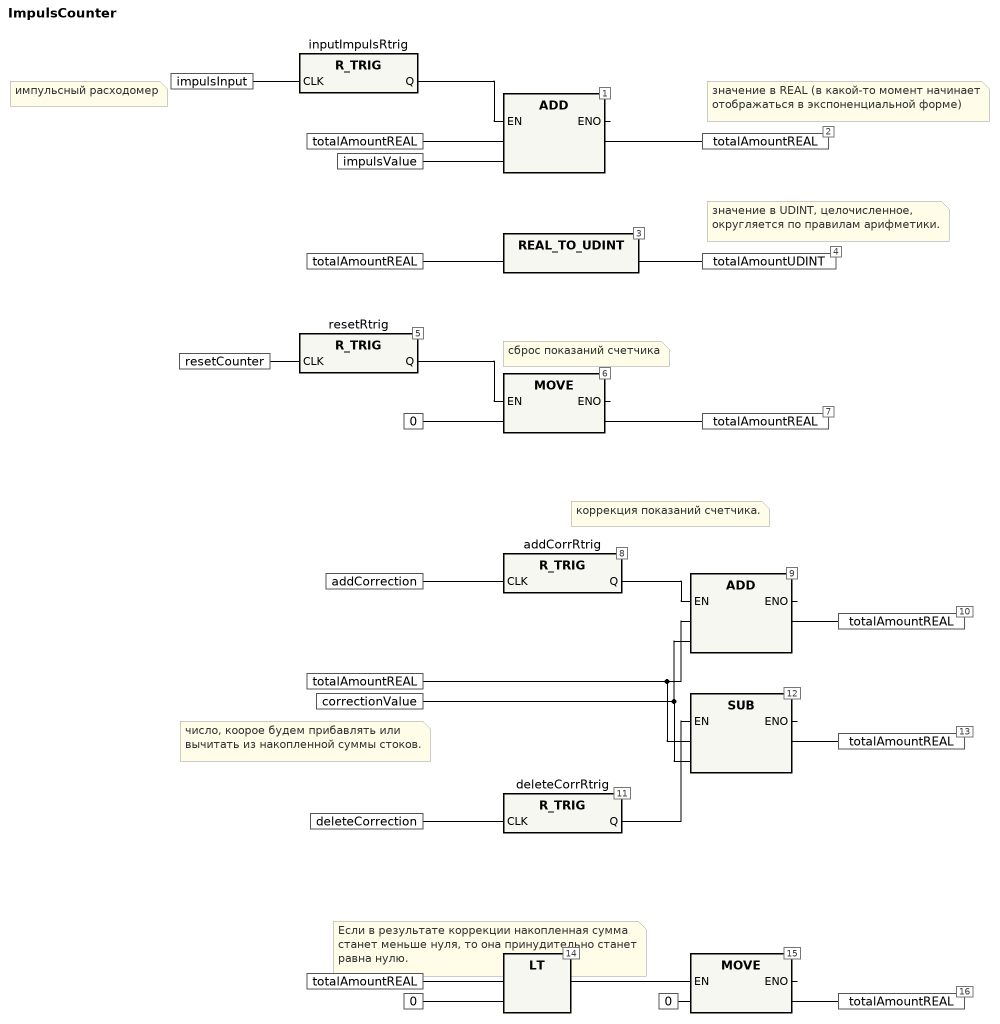
_CFC_ (* Continuous Function Chart, elements in execution order *)
(* импульсный расходомер *)
(* сброс показаний счетчика *)
(* значение в REAL (в какой-то момент начинает / отображаться в экспоненциальной форме) *)
(* значение в UDINT, целочисленное, / округляется по правилам арифметики. *)
(* Если в результате коррекции накопленная сумма станет меньше нуля, то она принудительно станет равна нулю. *)
(* коррекция показаний счетчика. *)
(* число, коорое будем прибавлять или / вычитать из накопленной суммы стоков. *)
#0 inputImpulsRtrig:R_TRIG(CLK: impulsInput)
#1 ADD(EN: #0.Q, totalAmountREAL, impulsValue)
#2 totalAmountREAL <= #1
#3 REAL_TO_UDINT(totalAmountREAL)
#4 totalAmountUDINT <= #3
#5 resetRtrig:R_TRIG(CLK: resetCounter)
#6 MOVE(EN: #5.Q, 0)
#7 totalAmountREAL <= #6
#8 addCorrRtrig:R_TRIG(CLK: addCorrection)
#9 ADD(EN: #8.Q, totalAmountREAL, correctionValue)
#10 totalAmountREAL <= #9
#11 deleteCorrRtrig:R_TRIG(CLK: deleteCorrection)
#12 SUB(EN: #11.Q, totalAmountREAL, correctionValue)
#13 totalAmountREAL <= #12
#14 LT(totalAmountREAL, 0)
#15 MOVE(EN: #14, 0)
#16 totalAmountREAL <= #15
_END_CFC_
(* the same logic as Structured Text *)
(* импульсный расходомер *)
(* сброс показаний счетчика *)
(* значение в REAL (в какой-то момент начинает / отображаться в экспоненциальной форме) *)
(* значение в UDINT, целочисленное, / округляется по правилам арифметики. *)
(* Если в результате коррекции накопленная сумма станет меньше нуля, то она принудительно станет равна нулю. *)
(* коррекция показаний счетчика. *)
(* число, коорое будем прибавлять или / вычитать из накопленной суммы стоков. *)
inputImpulsRtrig(CLK := impulsInput);
IF inputImpulsRtrig.Q THEN totalAmountREAL := totalAmountREAL + impulsValue; END_IF;
totalAmountUDINT := REAL_TO_UDINT(totalAmountREAL);
resetRtrig(CLK := resetCounter);
IF resetRtrig.Q THEN totalAmountREAL := 0; END_IF;
addCorrRtrig(CLK := addCorrection);
IF addCorrRtrig.Q THEN totalAmountREAL := totalAmountREAL + correctionValue; END_IF;
deleteCorrRtrig(CLK := deleteCorrection);
IF deleteCorrRtrig.Q THEN totalAmountREAL := totalAmountREAL - correctionValue; END_IF;
IF totalAmountREAL < 0 THEN totalAmountREAL := 0; END_IF;
END_FUNCTION_BLOCK

(* POU ManualTwoPumpManager, CFC *)
FUNCTION_BLOCK ManualTwoPumpManager
VAR_INPUT
	startStopPump1: BOOL;		(*Сигнал на пуск/стоп первого насоса.*)
	startStopPump2: BOOL;		(*Сигнал на пуск/стоп второго насоса.*)
	alarmPump1: BOOL;		(*Сигнал "авария" на первом насосе.*)
	alarmPump2: BOOL;		(*Сигнал "авария" на втором насосе.*)
	alarmReset: BOOL;		(*Сброс аварии.*)
END_VAR
VAR_OUTPUT
	pump1ON: BOOL;		(*Выход на включение первого насоса.*)
	pump2ON: BOOL;		(*Выход на включение второго насоса.*)
END_VAR
VAR
	RtrigPump1: R_TRIG;		(*Включает первый насос по фронту сигнала на ручной пуск/стоп.*)
	FtrigPump1: F_TRIG;		(*Выключает первый насос по спаду сигнала на ручной пуск/стоп.*)
	RtrigPump2: R_TRIG;		(*Включает второй насос по фронту сигнала на ручной пуск/стоп.*)
	FtrigPump2: F_TRIG;		(*Выключает второй насос по спаду сигнала на ручной пуск/стоп.*)
	RSpump1: RS;		(*RS-триггер нормального включения первого насоса*)
	RSpump2: RS;		(*RS-триггер нормального включения второго насоса*)
	pump1NormalON: BOOL;		(*Сигнал нормального (неаварийного) включения первого насоса.*)
	pump2NormalON: BOOL;		(*Сигнал нормального (неаварийного) включения второго насоса.*)
	pump2EmergencyON: BOOL;		(*Сигнал аварийного включения второго насоса (при аварии первого).*)
	pump1EmergencyON: BOOL;		(*Сигнал аварийного включения первого насоса (при аварии второго).*)
	alarmPump1RStrig: RS;		(*Триггер аварии первого насоса.*)
	alarmPump2RStrig: RS;		(*Триггер аварии второго насоса.*)
	TONtoOnPump1: TON;		(*Таймер задержки включения первого насоса, на переключение контакторов при аварийном переключении.
			Жестко задано 1 секунда.*)
	TONtoOnPump2: TON;		(*Таймер задержки включения второго насоса, на переключение контакторов при аварийном переключении.
						Жестко задано 1 секунда.*)
END_VAR
VAR (* helpers for the ST form of the networks *)
	_t119 : BOOL;
END_VAR
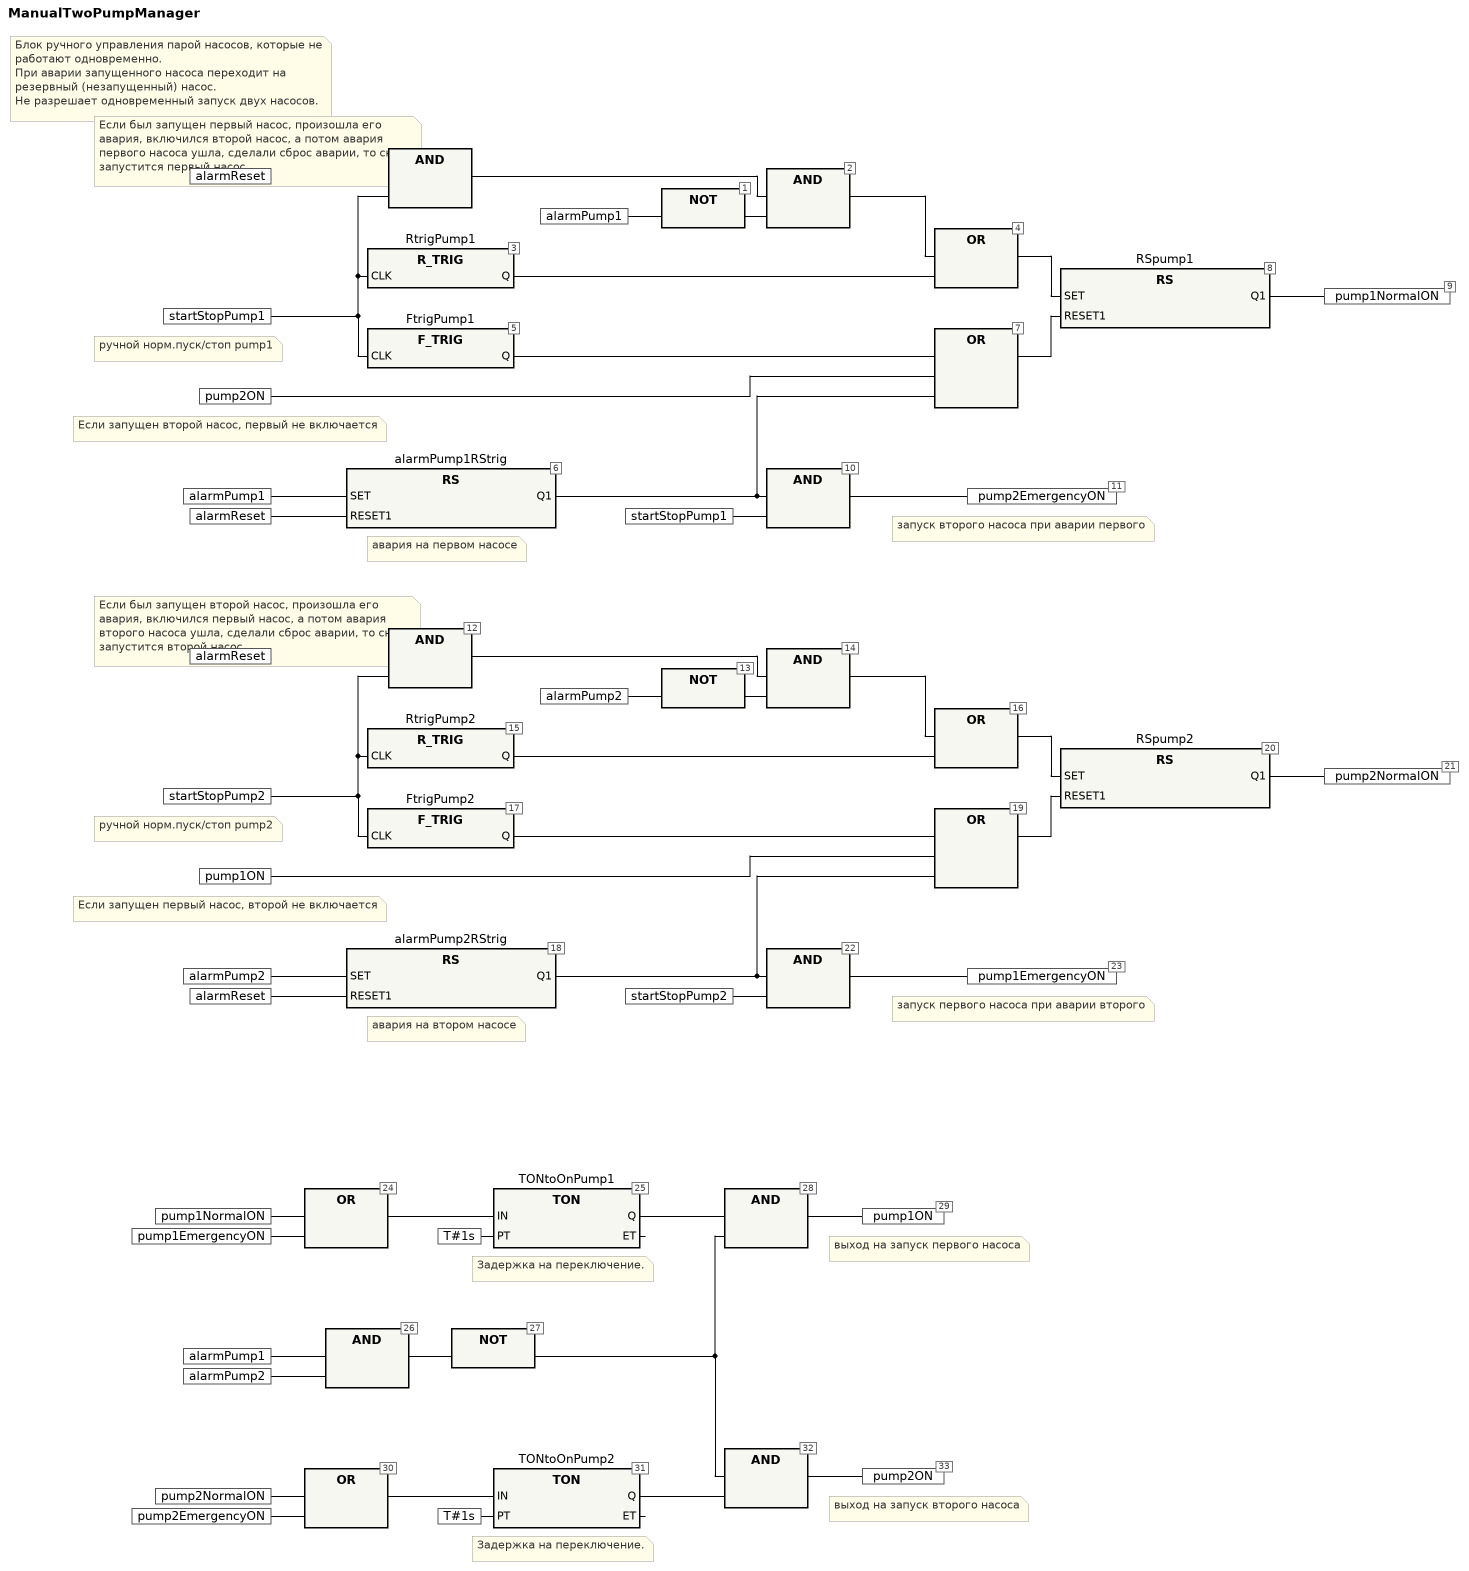
_CFC_ (* Continuous Function Chart, elements in execution order *)
(* Задержка на переключение. *)
(* Задержка на переключение. *)
(* выход на запуск второго насоса *)
(* выход на запуск первого насоса *)
(* запуск первого насоса при аварии второго *)
(* Если запущен первый насос, второй не включается *)
(* авария на втором насосе *)
(* ручной норм.пуск/стоп pump2 *)
(* ручной норм.пуск/стоп pump1 *)
(* запуск второго насоса при аварии первого *)
(* Если запущен второй насос, первый не включается *)
(* авария на первом насосе *)
(* Блок ручного управления парой насосов, которые не работают одновременно. / При аварии запущенного насоса переходит на резервный (незапущенный) насос. / Не разрешает одновременный запуск двух насосов. *)
(* Если был запущен первый насос, произошла его авария, включился второй насос, а потом авария первого насоса ушла, сделали сброс аварии, то снова запустится первый насос. *)
(* Если был запущен второй насос, произошла его авария, включился первый насос, а потом авария второго насоса ушла, сделали сброс аварии, то снова запустится второй насос. *)
#0 AND(alarmReset, startStopPump1)
#1 NOT(alarmPump1)
#2 AND(#0, #1)
#3 RtrigPump1:R_TRIG(CLK: startStopPump1)
#4 OR(#2, #3.Q)
#5 FtrigPump1:F_TRIG(CLK: startStopPump1)
#6 alarmPump1RStrig:RS(SET: alarmPump1, RESET1: alarmReset)
#7 OR(#5.Q, pump2ON, #6.Q1)
#8 RSpump1:RS(SET: #4, RESET1: #7)
#9 pump1NormalON <= #8.Q1
#10 AND(#6.Q1, startStopPump1)
#11 pump2EmergencyON <= #10
#12 AND(alarmReset, startStopPump2)
#13 NOT(alarmPump2)
#14 AND(#12, #13)
#15 RtrigPump2:R_TRIG(CLK: startStopPump2)
#16 OR(#14, #15.Q)
#17 FtrigPump2:F_TRIG(CLK: startStopPump2)
#18 alarmPump2RStrig:RS(SET: alarmPump2, RESET1: alarmReset)
#19 OR(#17.Q, pump1ON, #18.Q1)
#20 RSpump2:RS(SET: #16, RESET1: #19)
#21 pump2NormalON <= #20.Q1
#22 AND(#18.Q1, startStopPump2)
#23 pump1EmergencyON <= #22
#24 OR(pump1NormalON, pump1EmergencyON)
#25 TONtoOnPump1:TON(IN: #24, PT: T#1s)
#26 AND(alarmPump1, alarmPump2)
#27 NOT(#26)
#28 AND(#25.Q, #27)
#29 pump1ON <= #28
#30 OR(pump2NormalON, pump2EmergencyON)
#31 TONtoOnPump2:TON(IN: #30, PT: T#1s)
#32 AND(#27, #31.Q)
#33 pump2ON <= #32
_END_CFC_
(* the same logic as Structured Text *)
(* Задержка на переключение. *)
(* Задержка на переключение. *)
(* выход на запуск второго насоса *)
(* выход на запуск первого насоса *)
(* запуск первого насоса при аварии второго *)
(* Если запущен первый насос, второй не включается *)
(* авария на втором насосе *)
(* ручной норм.пуск/стоп pump2 *)
(* ручной норм.пуск/стоп pump1 *)
(* запуск второго насоса при аварии первого *)
(* Если запущен второй насос, первый не включается *)
(* авария на первом насосе *)
(* Блок ручного управления парой насосов, которые не работают одновременно. / При аварии запущенного насоса переходит на резервный (незапущенный) насос. / Не разрешает одновременный запуск двух насосов. *)
(* Если был запущен первый насос, произошла его авария, включился второй насос, а потом авария первого насоса ушла, сделали сброс аварии, то снова запустится первый насос. *)
(* Если был запущен второй насос, произошла его авария, включился первый насос, а потом авария второго насоса ушла, сделали сброс аварии, то снова запустится второй насос. *)
RtrigPump1(CLK := startStopPump1);
FtrigPump1(CLK := startStopPump1);
alarmPump1RStrig(SET := alarmPump1, RESET1 := alarmReset);
RSpump1(SET := ((alarmReset AND startStopPump1) AND NOT alarmPump1) OR RtrigPump1.Q, RESET1 := FtrigPump1.Q OR pump2ON OR alarmPump1RStrig.Q1);
pump1NormalON := RSpump1.Q1;
pump2EmergencyON := alarmPump1RStrig.Q1 AND startStopPump1;
RtrigPump2(CLK := startStopPump2);
FtrigPump2(CLK := startStopPump2);
alarmPump2RStrig(SET := alarmPump2, RESET1 := alarmReset);
RSpump2(SET := ((alarmReset AND startStopPump2) AND NOT alarmPump2) OR RtrigPump2.Q, RESET1 := FtrigPump2.Q OR pump1ON OR alarmPump2RStrig.Q1);
pump2NormalON := RSpump2.Q1;
pump1EmergencyON := alarmPump2RStrig.Q1 AND startStopPump2;
TONtoOnPump1(IN := pump1NormalON OR pump1EmergencyON, PT := T#1s);
_t119 := NOT (alarmPump1 AND alarmPump2);
pump1ON := TONtoOnPump1.Q AND _t119;
TONtoOnPump2(IN := pump2NormalON OR pump2EmergencyON, PT := T#1s);
pump2ON := _t119 AND TONtoOnPump2.Q;
END_FUNCTION_BLOCK
